(* Logix 5000 project; controller reports 1756-L63 rev 20.15; software revision 20.04; part 15 of 52 *)

        [677].log_data[17].valid := 1, [677].log_data[18].valid := 1, [677].log_data[19].valid := 1, [677].time.Year := 2023, [677].time.Month := 1, [677].time.Day := 12, [677].time.Minute := 49, [677].time.Second := 59, [678].log_data[0].min := 1.0, [678].log_data[0].max := 1.0, [678].log_data[0].total := 300.0, [678].log_data[0].time := 300.0, [678].log_data[0].minminute := 50, [678].log_data[0].maxminute := 50, [678].log_data[0].valid := 1, [678].log_data[1].valid := 1, [678].log_data[2].valid := 1, [678].log_data[3].valid := 1, [678].log_data[4].valid := 1, [678].log_data[5].valid := 1, [678].log_data[6].valid := 1, [678].log_data[7].valid := 1, [678].log_data[8].valid := 1, [678].log_data[9].valid := 1, [678].log_data[10].valid := 1, [678].log_data[11].valid := 1, [678].log_data[12].valid := 1, [678].log_data[13].valid := 1, [678].log_data[14].valid := 1, [678].log_data[15].valid := 1, [678].log_data[16].valid := 1, [678].log_data[17].valid := 1, [678].log_data[18].valid := 1, [678].log_data[19].valid := 1, [678].time.Year := 2023, [678].time.Month := 1, [678].time.Day := 12, [678].time.Minute := 54, [678].time.Second := 59, [679].log_data[0].min := 1.0, [679].log_data[0].max := 1.0, [679].log_data[0].total := 300.0, [679].log_data[0].time := 300.0, [679].log_data[0].minminute := 55, [679].log_data[0].maxminute := 55, [679].log_data[0].valid := 1, [679].log_data[1].valid := 1, [679].log_data[2].valid := 1, [679].log_data[3].valid := 1, [679].log_data[4].valid := 1, [679].log_data[5].valid := 1, [679].log_data[6].valid := 1, [679].log_data[7].valid := 1, [679].log_data[8].valid := 1, [679].log_data[9].valid := 1, [679].log_data[10].valid := 1, [679].log_data[11].valid := 1, [679].log_data[12].valid := 1, [679].log_data[13].valid := 1, [679].log_data[14].valid := 1,
        [679].log_data[15].valid := 1, [679].log_data[16].valid := 1, [679].log_data[17].valid := 1, [679].log_data[18].valid := 1, [679].log_data[19].valid := 1, [679].time.Year := 2023, [679].time.Month := 1, [679].time.Day := 12, [679].time.Minute := 59, [679].time.Second := 59, [680].log_data[0].min := 1.0, [680].log_data[0].max := 1.0, [680].log_data[0].total := 299.5, [680].log_data[0].time := 299.5, [680].log_data[0].valid := 1, [680].log_data[1].valid := 1, [680].log_data[2].valid := 1, [680].log_data[3].valid := 1, [680].log_data[4].valid := 1, [680].log_data[5].valid := 1, [680].log_data[6].valid := 1, [680].log_data[7].valid := 1, [680].log_data[8].valid := 1, [680].log_data[9].valid := 1, [680].log_data[10].valid := 1, [680].log_data[11].valid := 1, [680].log_data[12].valid := 1, [680].log_data[13].valid := 1, [680].log_data[14].valid := 1, [680].log_data[15].valid := 1, [680].log_data[16].valid := 1, [680].log_data[17].valid := 1, [680].log_data[18].valid := 1, [680].log_data[19].valid := 1, [680].time.Year := 2023, [680].time.Month := 1, [680].time.Day := 12, [680].time.Hour := 1, [680].time.Minute := 4, [680].time.Second := 59, [681].log_data[0].min := 1.0, [681].log_data[0].max := 1.0, [681].log_data[0].total := 300.0, [681].log_data[0].time := 300.0, [681].log_data[0].minminute := 5, [681].log_data[0].maxminute := 5, [681].log_data[0].valid := 1, [681].log_data[1].valid := 1, [681].log_data[2].valid := 1, [681].log_data[3].valid := 1, [681].log_data[4].valid := 1, [681].log_data[5].valid := 1, [681].log_data[6].valid := 1, [681].log_data[7].valid := 1, [681].log_data[8].valid := 1, [681].log_data[9].valid := 1, [681].log_data[10].valid := 1, [681].log_data[11].valid := 1, [681].log_data[12].valid := 1, [681].log_data[13].valid := 1,
        [681].log_data[14].valid := 1, [681].log_data[15].valid := 1, [681].log_data[16].valid := 1, [681].log_data[17].valid := 1, [681].log_data[18].valid := 1, [681].log_data[19].valid := 1, [681].time.Year := 2023, [681].time.Month := 1, [681].time.Day := 12, [681].time.Hour := 1, [681].time.Minute := 9, [681].time.Second := 59, [682].log_data[0].min := 1.0, [682].log_data[0].max := 1.0, [682].log_data[0].total := 300.0, [682].log_data[0].time := 300.0, [682].log_data[0].minminute := 10, [682].log_data[0].maxminute := 10, [682].log_data[0].valid := 1, [682].log_data[1].valid := 1, [682].log_data[2].valid := 1, [682].log_data[3].valid := 1, [682].log_data[4].valid := 1, [682].log_data[5].valid := 1, [682].log_data[6].valid := 1, [682].log_data[7].valid := 1, [682].log_data[8].valid := 1, [682].log_data[9].valid := 1, [682].log_data[10].valid := 1, [682].log_data[11].valid := 1, [682].log_data[12].valid := 1, [682].log_data[13].valid := 1, [682].log_data[14].valid := 1, [682].log_data[15].valid := 1, [682].log_data[16].valid := 1, [682].log_data[17].valid := 1, [682].log_data[18].valid := 1, [682].log_data[19].valid := 1, [682].time.Year := 2023, [682].time.Month := 1, [682].time.Day := 12, [682].time.Hour := 1, [682].time.Minute := 14, [682].time.Second := 59, [683].log_data[0].min := 1.0, [683].log_data[0].max := 1.0, [683].log_data[0].total := 300.0, [683].log_data[0].time := 300.0, [683].log_data[0].minminute := 15, [683].log_data[0].maxminute := 15, [683].log_data[0].valid := 1, [683].log_data[1].valid := 1, [683].log_data[2].valid := 1, [683].log_data[3].valid := 1, [683].log_data[4].valid := 1, [683].log_data[5].valid := 1, [683].log_data[6].valid := 1, [683].log_data[7].valid := 1, [683].log_data[8].valid := 1, [683].log_data[9].valid := 1,
        [683].log_data[10].valid := 1, [683].log_data[11].valid := 1, [683].log_data[12].valid := 1, [683].log_data[13].valid := 1, [683].log_data[14].valid := 1, [683].log_data[15].valid := 1, [683].log_data[16].valid := 1, [683].log_data[17].valid := 1, [683].log_data[18].valid := 1, [683].log_data[19].valid := 1, [683].time.Year := 2023, [683].time.Month := 1, [683].time.Day := 12, [683].time.Hour := 1, [683].time.Minute := 19, [683].time.Second := 59, [684].log_data[0].min := 1.0, [684].log_data[0].max := 1.0, [684].log_data[0].total := 300.0, [684].log_data[0].time := 300.0, [684].log_data[0].minminute := 20, [684].log_data[0].maxminute := 20, [684].log_data[0].valid := 1, [684].log_data[1].valid := 1, [684].log_data[2].valid := 1, [684].log_data[3].valid := 1, [684].log_data[4].valid := 1, [684].log_data[5].valid := 1, [684].log_data[6].valid := 1, [684].log_data[7].valid := 1, [684].log_data[8].valid := 1, [684].log_data[9].valid := 1, [684].log_data[10].valid := 1, [684].log_data[11].valid := 1, [684].log_data[12].valid := 1, [684].log_data[13].valid := 1, [684].log_data[14].valid := 1, [684].log_data[15].valid := 1, [684].log_data[16].valid := 1, [684].log_data[17].valid := 1, [684].log_data[18].valid := 1, [684].log_data[19].valid := 1, [684].time.Year := 2023, [684].time.Month := 1, [684].time.Day := 12, [684].time.Hour := 1, [684].time.Minute := 24, [684].time.Second := 59, [685].log_data[0].min := 1.0, [685].log_data[0].max := 1.0, [685].log_data[0].total := 300.0, [685].log_data[0].time := 300.0, [685].log_data[0].minminute := 25, [685].log_data[0].maxminute := 25, [685].log_data[0].valid := 1, [685].log_data[1].valid := 1, [685].log_data[2].valid := 1, [685].log_data[3].valid := 1, [685].log_data[4].valid := 1, [685].log_data[5].valid := 1,
        [685].log_data[6].valid := 1, [685].log_data[7].valid := 1, [685].log_data[8].valid := 1, [685].log_data[9].valid := 1, [685].log_data[10].valid := 1, [685].log_data[11].valid := 1, [685].log_data[12].valid := 1, [685].log_data[13].valid := 1, [685].log_data[14].valid := 1, [685].log_data[15].valid := 1, [685].log_data[16].valid := 1, [685].log_data[17].valid := 1, [685].log_data[18].valid := 1, [685].log_data[19].valid := 1, [685].time.Year := 2023, [685].time.Month := 1, [685].time.Day := 12, [685].time.Hour := 1, [685].time.Minute := 29, [685].time.Second := 59, [686].log_data[0].min := 1.0, [686].log_data[0].max := 1.0, [686].log_data[0].total := 300.0, [686].log_data[0].time := 300.0, [686].log_data[0].minminute := 30, [686].log_data[0].maxminute := 30, [686].log_data[0].valid := 1, [686].log_data[1].valid := 1, [686].log_data[2].valid := 1, [686].log_data[3].valid := 1, [686].log_data[4].valid := 1, [686].log_data[5].valid := 1, [686].log_data[6].valid := 1, [686].log_data[7].valid := 1, [686].log_data[8].valid := 1, [686].log_data[9].valid := 1, [686].log_data[10].valid := 1, [686].log_data[11].valid := 1, [686].log_data[12].valid := 1, [686].log_data[13].valid := 1, [686].log_data[14].valid := 1, [686].log_data[15].valid := 1, [686].log_data[16].valid := 1, [686].log_data[17].valid := 1, [686].log_data[18].valid := 1, [686].log_data[19].valid := 1, [686].time.Year := 2023, [686].time.Month := 1, [686].time.Day := 12, [686].time.Hour := 1, [686].time.Minute := 34, [686].time.Second := 59, [687].log_data[0].min := 1.0, [687].log_data[0].max := 1.0, [687].log_data[0].total := 300.0, [687].log_data[0].time := 300.0, [687].log_data[0].minminute := 35, [687].log_data[0].maxminute := 35, [687].log_data[0].valid := 1, [687].log_data[1].valid := 1,
        [687].log_data[2].valid := 1, [687].log_data[3].valid := 1, [687].log_data[4].valid := 1, [687].log_data[5].valid := 1, [687].log_data[6].valid := 1, [687].log_data[7].valid := 1, [687].log_data[8].valid := 1, [687].log_data[9].valid := 1, [687].log_data[10].valid := 1, [687].log_data[11].valid := 1, [687].log_data[12].valid := 1, [687].log_data[13].valid := 1, [687].log_data[14].valid := 1, [687].log_data[15].valid := 1, [687].log_data[16].valid := 1, [687].log_data[17].valid := 1, [687].log_data[18].valid := 1, [687].log_data[19].valid := 1, [687].time.Year := 2023, [687].time.Month := 1, [687].time.Day := 12, [687].time.Hour := 1, [687].time.Minute := 39, [687].time.Second := 59, [688].log_data[0].min := 1.0, [688].log_data[0].max := 1.0, [688].log_data[0].total := 300.0, [688].log_data[0].time := 300.0, [688].log_data[0].minminute := 40, [688].log_data[0].maxminute := 40, [688].log_data[0].valid := 1, [688].log_data[1].valid := 1, [688].log_data[2].valid := 1, [688].log_data[3].valid := 1, [688].log_data[4].valid := 1, [688].log_data[5].valid := 1, [688].log_data[6].valid := 1, [688].log_data[7].valid := 1, [688].log_data[8].valid := 1, [688].log_data[9].valid := 1, [688].log_data[10].valid := 1, [688].log_data[11].valid := 1, [688].log_data[12].valid := 1, [688].log_data[13].valid := 1, [688].log_data[14].valid := 1, [688].log_data[15].valid := 1, [688].log_data[16].valid := 1, [688].log_data[17].valid := 1, [688].log_data[18].valid := 1, [688].log_data[19].valid := 1, [688].time.Year := 2023, [688].time.Month := 1, [688].time.Day := 12, [688].time.Hour := 1, [688].time.Minute := 44, [688].time.Second := 59, [689].log_data[0].min := 1.0, [689].log_data[0].max := 1.0, [689].log_data[0].total := 300.0, [689].log_data[0].time := 300.0,
        [689].log_data[0].minminute := 45, [689].log_data[0].maxminute := 45, [689].log_data[0].valid := 1, [689].log_data[1].valid := 1, [689].log_data[2].valid := 1, [689].log_data[3].valid := 1, [689].log_data[4].valid := 1, [689].log_data[5].valid := 1, [689].log_data[6].valid := 1, [689].log_data[7].valid := 1, [689].log_data[8].valid := 1, [689].log_data[9].valid := 1, [689].log_data[10].valid := 1, [689].log_data[11].valid := 1, [689].log_data[12].valid := 1, [689].log_data[13].valid := 1, [689].log_data[14].valid := 1, [689].log_data[15].valid := 1, [689].log_data[16].valid := 1, [689].log_data[17].valid := 1, [689].log_data[18].valid := 1, [689].log_data[19].valid := 1, [689].time.Year := 2023, [689].time.Month := 1, [689].time.Day := 12, [689].time.Hour := 1, [689].time.Minute := 49, [689].time.Second := 59, [690].log_data[0].min := 1.0, [690].log_data[0].max := 1.0, [690].log_data[0].total := 300.0, [690].log_data[0].time := 300.0, [690].log_data[0].minminute := 50, [690].log_data[0].maxminute := 50, [690].log_data[0].valid := 1, [690].log_data[1].valid := 1, [690].log_data[2].valid := 1, [690].log_data[3].valid := 1, [690].log_data[4].valid := 1, [690].log_data[5].valid := 1, [690].log_data[6].valid := 1, [690].log_data[7].valid := 1, [690].log_data[8].valid := 1, [690].log_data[9].valid := 1, [690].log_data[10].valid := 1, [690].log_data[11].valid := 1, [690].log_data[12].valid := 1, [690].log_data[13].valid := 1, [690].log_data[14].valid := 1, [690].log_data[15].valid := 1, [690].log_data[16].valid := 1, [690].log_data[17].valid := 1, [690].log_data[18].valid := 1, [690].log_data[19].valid := 1, [690].time.Year := 2023, [690].time.Month := 1, [690].time.Day := 12, [690].time.Hour := 1, [690].time.Minute := 54, [690].time.Second := 59,
        [691].log_data[0].min := 1.0, [691].log_data[0].max := 1.0, [691].log_data[0].total := 300.0, [691].log_data[0].time := 300.0, [691].log_data[0].minminute := 55, [691].log_data[0].maxminute := 55, [691].log_data[0].valid := 1, [691].log_data[1].valid := 1, [691].log_data[2].valid := 1, [691].log_data[3].valid := 1, [691].log_data[4].valid := 1, [691].log_data[5].valid := 1, [691].log_data[6].valid := 1, [691].log_data[7].valid := 1, [691].log_data[8].valid := 1, [691].log_data[9].valid := 1, [691].log_data[10].valid := 1, [691].log_data[11].valid := 1, [691].log_data[12].valid := 1, [691].log_data[13].valid := 1, [691].log_data[14].valid := 1, [691].log_data[15].valid := 1, [691].log_data[16].valid := 1, [691].log_data[17].valid := 1, [691].log_data[18].valid := 1, [691].log_data[19].valid := 1, [691].time.Year := 2023, [691].time.Month := 1, [691].time.Day := 12, [691].time.Hour := 1, [691].time.Minute := 59, [691].time.Second := 59, [692].log_data[0].min := 1.0, [692].log_data[0].max := 1.0, [692].log_data[0].total := 300.0, [692].log_data[0].time := 300.0, [692].log_data[0].valid := 1, [692].log_data[1].valid := 1, [692].log_data[2].valid := 1, [692].log_data[3].valid := 1, [692].log_data[4].valid := 1, [692].log_data[5].valid := 1, [692].log_data[6].valid := 1, [692].log_data[7].valid := 1, [692].log_data[8].valid := 1, [692].log_data[9].valid := 1, [692].log_data[10].valid := 1, [692].log_data[11].valid := 1, [692].log_data[12].valid := 1, [692].log_data[13].valid := 1, [692].log_data[14].valid := 1, [692].log_data[15].valid := 1, [692].log_data[16].valid := 1, [692].log_data[17].valid := 1, [692].log_data[18].valid := 1, [692].log_data[19].valid := 1, [692].time.Year := 2023, [692].time.Month := 1, [692].time.Day := 12, [692].time.Hour := 2,
        [692].time.Minute := 4, [692].time.Second := 59, [693].log_data[0].min := 1.0, [693].log_data[0].max := 1.0, [693].log_data[0].total := 300.0, [693].log_data[0].time := 300.0, [693].log_data[0].minminute := 5, [693].log_data[0].maxminute := 5, [693].log_data[0].valid := 1, [693].log_data[1].valid := 1, [693].log_data[2].valid := 1, [693].log_data[3].valid := 1, [693].log_data[4].valid := 1, [693].log_data[5].valid := 1, [693].log_data[6].valid := 1, [693].log_data[7].valid := 1, [693].log_data[8].valid := 1, [693].log_data[9].valid := 1, [693].log_data[10].valid := 1, [693].log_data[11].valid := 1, [693].log_data[12].valid := 1, [693].log_data[13].valid := 1, [693].log_data[14].valid := 1, [693].log_data[15].valid := 1, [693].log_data[16].valid := 1, [693].log_data[17].valid := 1, [693].log_data[18].valid := 1, [693].log_data[19].valid := 1, [693].time.Year := 2023, [693].time.Month := 1, [693].time.Day := 12, [693].time.Hour := 2, [693].time.Minute := 9, [693].time.Second := 59, [694].log_data[0].min := 1.0, [694].log_data[0].max := 1.0, [694].log_data[0].total := 300.0, [694].log_data[0].time := 300.0, [694].log_data[0].minminute := 10, [694].log_data[0].maxminute := 10, [694].log_data[0].valid := 1, [694].log_data[1].valid := 1, [694].log_data[2].valid := 1, [694].log_data[3].valid := 1, [694].log_data[4].valid := 1, [694].log_data[5].valid := 1, [694].log_data[6].valid := 1, [694].log_data[7].valid := 1, [694].log_data[8].valid := 1, [694].log_data[9].valid := 1, [694].log_data[10].valid := 1, [694].log_data[11].valid := 1, [694].log_data[12].valid := 1, [694].log_data[13].valid := 1, [694].log_data[14].valid := 1, [694].log_data[15].valid := 1, [694].log_data[16].valid := 1, [694].log_data[17].valid := 1, [694].log_data[18].valid := 1, [694].log_data[19].valid := 1,
        [694].time.Year := 2023, [694].time.Month := 1, [694].time.Day := 12, [694].time.Hour := 2, [694].time.Minute := 14, [694].time.Second := 59, [695].log_data[0].min := 1.0, [695].log_data[0].max := 1.0, [695].log_data[0].total := 300.0, [695].log_data[0].time := 300.0, [695].log_data[0].minminute := 15, [695].log_data[0].maxminute := 15, [695].log_data[0].valid := 1, [695].log_data[1].valid := 1, [695].log_data[2].valid := 1, [695].log_data[3].valid := 1, [695].log_data[4].valid := 1, [695].log_data[5].valid := 1, [695].log_data[6].valid := 1, [695].log_data[7].valid := 1, [695].log_data[8].valid := 1, [695].log_data[9].valid := 1, [695].log_data[10].valid := 1, [695].log_data[11].valid := 1, [695].log_data[12].valid := 1, [695].log_data[13].valid := 1, [695].log_data[14].valid := 1, [695].log_data[15].valid := 1, [695].log_data[16].valid := 1, [695].log_data[17].valid := 1, [695].log_data[18].valid := 1, [695].log_data[19].valid := 1, [695].time.Year := 2023, [695].time.Month := 1, [695].time.Day := 12, [695].time.Hour := 2, [695].time.Minute := 19, [695].time.Second := 59, [696].log_data[0].min := 1.0, [696].log_data[0].max := 1.0, [696].log_data[0].total := 300.0, [696].log_data[0].time := 300.0, [696].log_data[0].minminute := 20, [696].log_data[0].maxminute := 20, [696].log_data[0].valid := 1, [696].log_data[1].valid := 1, [696].log_data[2].valid := 1, [696].log_data[3].valid := 1, [696].log_data[4].valid := 1, [696].log_data[5].valid := 1, [696].log_data[6].valid := 1, [696].log_data[7].valid := 1, [696].log_data[8].valid := 1, [696].log_data[9].valid := 1, [696].log_data[10].valid := 1, [696].log_data[11].valid := 1, [696].log_data[12].valid := 1, [696].log_data[13].valid := 1, [696].log_data[14].valid := 1, [696].log_data[15].valid := 1,
        [696].log_data[16].valid := 1, [696].log_data[17].valid := 1, [696].log_data[18].valid := 1, [696].log_data[19].valid := 1, [696].time.Year := 2023, [696].time.Month := 1, [696].time.Day := 12, [696].time.Hour := 2, [696].time.Minute := 24, [696].time.Second := 59, [697].log_data[0].min := 1.0, [697].log_data[0].max := 1.0, [697].log_data[0].total := 300.0, [697].log_data[0].time := 300.0, [697].log_data[0].minminute := 25, [697].log_data[0].maxminute := 25, [697].log_data[0].valid := 1, [697].log_data[1].valid := 1, [697].log_data[2].valid := 1, [697].log_data[3].valid := 1, [697].log_data[4].valid := 1, [697].log_data[5].valid := 1, [697].log_data[6].valid := 1, [697].log_data[7].valid := 1, [697].log_data[8].valid := 1, [697].log_data[9].valid := 1, [697].log_data[10].valid := 1, [697].log_data[11].valid := 1, [697].log_data[12].valid := 1, [697].log_data[13].valid := 1, [697].log_data[14].valid := 1, [697].log_data[15].valid := 1, [697].log_data[16].valid := 1, [697].log_data[17].valid := 1, [697].log_data[18].valid := 1, [697].log_data[19].valid := 1, [697].time.Year := 2023, [697].time.Month := 1, [697].time.Day := 12, [697].time.Hour := 2, [697].time.Minute := 29, [697].time.Second := 59, [698].log_data[0].min := 1.0, [698].log_data[0].max := 1.0, [698].log_data[0].total := 300.0, [698].log_data[0].time := 300.0, [698].log_data[0].minminute := 30, [698].log_data[0].maxminute := 30, [698].log_data[0].valid := 1, [698].log_data[1].valid := 1, [698].log_data[2].valid := 1, [698].log_data[3].valid := 1, [698].log_data[4].valid := 1, [698].log_data[5].valid := 1, [698].log_data[6].valid := 1, [698].log_data[7].valid := 1, [698].log_data[8].valid := 1, [698].log_data[9].valid := 1, [698].log_data[10].valid := 1, [698].log_data[11].valid := 1,
        [698].log_data[12].valid := 1, [698].log_data[13].valid := 1, [698].log_data[14].valid := 1, [698].log_data[15].valid := 1, [698].log_data[16].valid := 1, [698].log_data[17].valid := 1, [698].log_data[18].valid := 1, [698].log_data[19].valid := 1, [698].time.Year := 2023, [698].time.Month := 1, [698].time.Day := 12, [698].time.Hour := 2, [698].time.Minute := 34, [698].time.Second := 59, [699].log_data[0].min := 1.0, [699].log_data[0].max := 1.0, [699].log_data[0].total := 300.0, [699].log_data[0].time := 300.0, [699].log_data[0].minminute := 35, [699].log_data[0].maxminute := 35, [699].log_data[0].valid := 1, [699].log_data[1].valid := 1, [699].log_data[2].valid := 1, [699].log_data[3].valid := 1, [699].log_data[4].valid := 1, [699].log_data[5].valid := 1, [699].log_data[6].valid := 1, [699].log_data[7].valid := 1, [699].log_data[8].valid := 1, [699].log_data[9].valid := 1, [699].log_data[10].valid := 1, [699].log_data[11].valid := 1, [699].log_data[12].valid := 1, [699].log_data[13].valid := 1, [699].log_data[14].valid := 1, [699].log_data[15].valid := 1, [699].log_data[16].valid := 1, [699].log_data[17].valid := 1, [699].log_data[18].valid := 1, [699].log_data[19].valid := 1, [699].time.Year := 2023, [699].time.Month := 1, [699].time.Day := 12, [699].time.Hour := 2, [699].time.Minute := 39, [699].time.Second := 59, [700].log_data[0].min := 1.0, [700].log_data[0].max := 1.0, [700].log_data[0].total := 300.0, [700].log_data[0].time := 300.0, [700].log_data[0].minminute := 40, [700].log_data[0].maxminute := 40, [700].log_data[0].valid := 1, [700].log_data[1].valid := 1, [700].log_data[2].valid := 1, [700].log_data[3].valid := 1, [700].log_data[4].valid := 1, [700].log_data[5].valid := 1, [700].log_data[6].valid := 1, [700].log_data[7].valid := 1,
        [700].log_data[8].valid := 1, [700].log_data[9].valid := 1, [700].log_data[10].valid := 1, [700].log_data[11].valid := 1, [700].log_data[12].valid := 1, [700].log_data[13].valid := 1, [700].log_data[14].valid := 1, [700].log_data[15].valid := 1, [700].log_data[16].valid := 1, [700].log_data[17].valid := 1, [700].log_data[18].valid := 1, [700].log_data[19].valid := 1, [700].time.Year := 2023, [700].time.Month := 1, [700].time.Day := 12, [700].time.Hour := 2, [700].time.Minute := 44, [700].time.Second := 59, [701].log_data[0].min := 1.0, [701].log_data[0].max := 1.0, [701].log_data[0].total := 300.0, [701].log_data[0].time := 300.0, [701].log_data[0].minminute := 45, [701].log_data[0].maxminute := 45, [701].log_data[0].valid := 1, [701].log_data[1].valid := 1, [701].log_data[2].valid := 1, [701].log_data[3].valid := 1, [701].log_data[4].valid := 1, [701].log_data[5].valid := 1, [701].log_data[6].valid := 1, [701].log_data[7].valid := 1, [701].log_data[8].valid := 1, [701].log_data[9].valid := 1, [701].log_data[10].valid := 1, [701].log_data[11].valid := 1, [701].log_data[12].valid := 1, [701].log_data[13].valid := 1, [701].log_data[14].valid := 1, [701].log_data[15].valid := 1, [701].log_data[16].valid := 1, [701].log_data[17].valid := 1, [701].log_data[18].valid := 1, [701].log_data[19].valid := 1, [701].time.Year := 2023, [701].time.Month := 1, [701].time.Day := 12, [701].time.Hour := 2, [701].time.Minute := 49, [701].time.Second := 59, [702].log_data[0].min := 1.0, [702].log_data[0].max := 1.0, [702].log_data[0].total := 300.0, [702].log_data[0].time := 300.0, [702].log_data[0].minminute := 50, [702].log_data[0].maxminute := 50, [702].log_data[0].valid := 1, [702].log_data[1].valid := 1, [702].log_data[2].valid := 1, [702].log_data[3].valid := 1,
        [702].log_data[4].valid := 1, [702].log_data[5].valid := 1, [702].log_data[6].valid := 1, [702].log_data[7].valid := 1, [702].log_data[8].valid := 1, [702].log_data[9].valid := 1, [702].log_data[10].valid := 1, [702].log_data[11].valid := 1, [702].log_data[12].valid := 1, [702].log_data[13].valid := 1, [702].log_data[14].valid := 1, [702].log_data[15].valid := 1, [702].log_data[16].valid := 1, [702].log_data[17].valid := 1, [702].log_data[18].valid := 1, [702].log_data[19].valid := 1, [702].time.Year := 2023, [702].time.Month := 1, [702].time.Day := 12, [702].time.Hour := 2, [702].time.Minute := 54, [702].time.Second := 59, [703].log_data[0].min := 1.0, [703].log_data[0].max := 1.0, [703].log_data[0].total := 300.0, [703].log_data[0].time := 300.0, [703].log_data[0].minminute := 55, [703].log_data[0].maxminute := 55, [703].log_data[0].valid := 1, [703].log_data[1].valid := 1, [703].log_data[2].valid := 1, [703].log_data[3].valid := 1, [703].log_data[4].valid := 1, [703].log_data[5].valid := 1, [703].log_data[6].valid := 1, [703].log_data[7].valid := 1, [703].log_data[8].valid := 1, [703].log_data[9].valid := 1, [703].log_data[10].valid := 1, [703].log_data[11].valid := 1, [703].log_data[12].valid := 1, [703].log_data[13].valid := 1, [703].log_data[14].valid := 1, [703].log_data[15].valid := 1, [703].log_data[16].valid := 1, [703].log_data[17].valid := 1, [703].log_data[18].valid := 1, [703].log_data[19].valid := 1, [703].time.Year := 2023, [703].time.Month := 1, [703].time.Day := 12, [703].time.Hour := 2, [703].time.Minute := 59, [703].time.Second := 59, [704].log_data[0].min := 1.0, [704].log_data[0].max := 1.0, [704].log_data[0].total := 300.0, [704].log_data[0].time := 300.0, [704].log_data[0].valid := 1, [704].log_data[1].valid := 1,
        [704].log_data[2].valid := 1, [704].log_data[3].valid := 1, [704].log_data[4].valid := 1, [704].log_data[5].valid := 1, [704].log_data[6].valid := 1, [704].log_data[7].valid := 1, [704].log_data[8].valid := 1, [704].log_data[9].valid := 1, [704].log_data[10].valid := 1, [704].log_data[11].valid := 1, [704].log_data[12].valid := 1, [704].log_data[13].valid := 1, [704].log_data[14].valid := 1, [704].log_data[15].valid := 1, [704].log_data[16].valid := 1, [704].log_data[17].valid := 1, [704].log_data[18].valid := 1, [704].log_data[19].valid := 1, [704].time.Year := 2023, [704].time.Month := 1, [704].time.Day := 12, [704].time.Hour := 3, [704].time.Minute := 4, [704].time.Second := 59, [705].log_data[0].min := 1.0, [705].log_data[0].max := 1.0, [705].log_data[0].total := 300.0, [705].log_data[0].time := 300.0, [705].log_data[0].minminute := 5, [705].log_data[0].maxminute := 5, [705].log_data[0].valid := 1, [705].log_data[1].valid := 1, [705].log_data[2].valid := 1, [705].log_data[3].valid := 1, [705].log_data[4].valid := 1, [705].log_data[5].valid := 1, [705].log_data[6].valid := 1, [705].log_data[7].valid := 1, [705].log_data[8].valid := 1, [705].log_data[9].valid := 1, [705].log_data[10].valid := 1, [705].log_data[11].valid := 1, [705].log_data[12].valid := 1, [705].log_data[13].valid := 1, [705].log_data[14].valid := 1, [705].log_data[15].valid := 1, [705].log_data[16].valid := 1, [705].log_data[17].valid := 1, [705].log_data[18].valid := 1, [705].log_data[19].valid := 1, [705].time.Year := 2023, [705].time.Month := 1, [705].time.Day := 12, [705].time.Hour := 3, [705].time.Minute := 9, [705].time.Second := 59, [706].log_data[0].min := 1.0, [706].log_data[0].max := 1.0, [706].log_data[0].total := 300.0, [706].log_data[0].time := 300.0,
        [706].log_data[0].minminute := 10, [706].log_data[0].maxminute := 10, [706].log_data[0].valid := 1, [706].log_data[1].valid := 1, [706].log_data[2].valid := 1, [706].log_data[3].valid := 1, [706].log_data[4].valid := 1, [706].log_data[5].valid := 1, [706].log_data[6].valid := 1, [706].log_data[7].valid := 1, [706].log_data[8].valid := 1, [706].log_data[9].valid := 1, [706].log_data[10].valid := 1, [706].log_data[11].valid := 1, [706].log_data[12].valid := 1, [706].log_data[13].valid := 1, [706].log_data[14].valid := 1, [706].log_data[15].valid := 1, [706].log_data[16].valid := 1, [706].log_data[17].valid := 1, [706].log_data[18].valid := 1, [706].log_data[19].valid := 1, [706].time.Year := 2023, [706].time.Month := 1, [706].time.Day := 12, [706].time.Hour := 3, [706].time.Minute := 14, [706].time.Second := 59, [707].log_data[0].min := 1.0, [707].log_data[0].max := 1.0, [707].log_data[0].total := 300.0, [707].log_data[0].time := 300.0, [707].log_data[0].minminute := 15, [707].log_data[0].maxminute := 15, [707].log_data[0].valid := 1, [707].log_data[1].valid := 1, [707].log_data[2].valid := 1, [707].log_data[3].valid := 1, [707].log_data[4].valid := 1, [707].log_data[5].valid := 1, [707].log_data[6].valid := 1, [707].log_data[7].valid := 1, [707].log_data[8].valid := 1, [707].log_data[9].valid := 1, [707].log_data[10].valid := 1, [707].log_data[11].valid := 1, [707].log_data[12].valid := 1, [707].log_data[13].valid := 1, [707].log_data[14].valid := 1, [707].log_data[15].valid := 1, [707].log_data[16].valid := 1, [707].log_data[17].valid := 1, [707].log_data[18].valid := 1, [707].log_data[19].valid := 1, [707].time.Year := 2023, [707].time.Month := 1, [707].time.Day := 12, [707].time.Hour := 3, [707].time.Minute := 19, [707].time.Second := 59,
        [708].log_data[0].min := 1.0, [708].log_data[0].max := 1.0, [708].log_data[0].total := 300.0, [708].log_data[0].time := 300.0, [708].log_data[0].minminute := 20, [708].log_data[0].maxminute := 20, [708].log_data[0].valid := 1, [708].log_data[1].valid := 1, [708].log_data[2].valid := 1, [708].log_data[3].valid := 1, [708].log_data[4].valid := 1, [708].log_data[5].valid := 1, [708].log_data[6].valid := 1, [708].log_data[7].valid := 1, [708].log_data[8].valid := 1, [708].log_data[9].valid := 1, [708].log_data[10].valid := 1, [708].log_data[11].valid := 1, [708].log_data[12].valid := 1, [708].log_data[13].valid := 1, [708].log_data[14].valid := 1, [708].log_data[15].valid := 1, [708].log_data[16].valid := 1, [708].log_data[17].valid := 1, [708].log_data[18].valid := 1, [708].log_data[19].valid := 1, [708].time.Year := 2023, [708].time.Month := 1, [708].time.Day := 12, [708].time.Hour := 3, [708].time.Minute := 24, [708].time.Second := 59, [709].log_data[0].min := 1.0, [709].log_data[0].max := 1.0, [709].log_data[0].total := 300.0, [709].log_data[0].time := 300.0, [709].log_data[0].minminute := 25, [709].log_data[0].maxminute := 25, [709].log_data[0].valid := 1, [709].log_data[1].valid := 1, [709].log_data[2].valid := 1, [709].log_data[3].valid := 1, [709].log_data[4].valid := 1, [709].log_data[5].valid := 1, [709].log_data[6].valid := 1, [709].log_data[7].valid := 1, [709].log_data[8].valid := 1, [709].log_data[9].valid := 1, [709].log_data[10].valid := 1, [709].log_data[11].valid := 1, [709].log_data[12].valid := 1, [709].log_data[13].valid := 1, [709].log_data[14].valid := 1, [709].log_data[15].valid := 1, [709].log_data[16].valid := 1, [709].log_data[17].valid := 1, [709].log_data[18].valid := 1, [709].log_data[19].valid := 1, [709].time.Year := 2023, [709].time.Month := 1,
        [709].time.Day := 12, [709].time.Hour := 3, [709].time.Minute := 29, [709].time.Second := 59, [710].log_data[0].min := 1.0, [710].log_data[0].max := 1.0, [710].log_data[0].total := 300.0, [710].log_data[0].time := 300.0, [710].log_data[0].minminute := 30, [710].log_data[0].maxminute := 30, [710].log_data[0].valid := 1, [710].log_data[1].valid := 1, [710].log_data[2].valid := 1, [710].log_data[3].valid := 1, [710].log_data[4].valid := 1, [710].log_data[5].valid := 1, [710].log_data[6].valid := 1, [710].log_data[7].valid := 1, [710].log_data[8].valid := 1, [710].log_data[9].valid := 1, [710].log_data[10].valid := 1, [710].log_data[11].valid := 1, [710].log_data[12].valid := 1, [710].log_data[13].valid := 1, [710].log_data[14].valid := 1, [710].log_data[15].valid := 1, [710].log_data[16].valid := 1, [710].log_data[17].valid := 1, [710].log_data[18].valid := 1, [710].log_data[19].valid := 1, [710].time.Year := 2023, [710].time.Month := 1, [710].time.Day := 12, [710].time.Hour := 3, [710].time.Minute := 34, [710].time.Second := 59, [711].log_data[0].min := 1.0, [711].log_data[0].max := 1.0, [711].log_data[0].total := 300.0, [711].log_data[0].time := 300.0, [711].log_data[0].minminute := 35, [711].log_data[0].maxminute := 35, [711].log_data[0].valid := 1, [711].log_data[1].valid := 1, [711].log_data[2].valid := 1, [711].log_data[3].valid := 1, [711].log_data[4].valid := 1, [711].log_data[5].valid := 1, [711].log_data[6].valid := 1, [711].log_data[7].valid := 1, [711].log_data[8].valid := 1, [711].log_data[9].valid := 1, [711].log_data[10].valid := 1, [711].log_data[11].valid := 1, [711].log_data[12].valid := 1, [711].log_data[13].valid := 1, [711].log_data[14].valid := 1, [711].log_data[15].valid := 1, [711].log_data[16].valid := 1, [711].log_data[17].valid := 1,
        [711].log_data[18].valid := 1, [711].log_data[19].valid := 1, [711].time.Year := 2023, [711].time.Month := 1, [711].time.Day := 12, [711].time.Hour := 3, [711].time.Minute := 39, [711].time.Second := 59, [712].log_data[0].min := 1.0, [712].log_data[0].max := 1.0, [712].log_data[0].total := 300.0, [712].log_data[0].time := 300.0, [712].log_data[0].minminute := 40, [712].log_data[0].maxminute := 40, [712].log_data[0].valid := 1, [712].log_data[1].valid := 1, [712].log_data[2].valid := 1, [712].log_data[3].valid := 1, [712].log_data[4].valid := 1, [712].log_data[5].valid := 1, [712].log_data[6].valid := 1, [712].log_data[7].valid := 1, [712].log_data[8].valid := 1, [712].log_data[9].valid := 1, [712].log_data[10].valid := 1, [712].log_data[11].valid := 1, [712].log_data[12].valid := 1, [712].log_data[13].valid := 1, [712].log_data[14].valid := 1, [712].log_data[15].valid := 1, [712].log_data[16].valid := 1, [712].log_data[17].valid := 1, [712].log_data[18].valid := 1, [712].log_data[19].valid := 1, [712].time.Year := 2023, [712].time.Month := 1, [712].time.Day := 12, [712].time.Hour := 3, [712].time.Minute := 44, [712].time.Second := 59, [713].log_data[0].min := 1.0, [713].log_data[0].max := 1.0, [713].log_data[0].total := 300.0, [713].log_data[0].time := 300.0, [713].log_data[0].minminute := 45, [713].log_data[0].maxminute := 45, [713].log_data[0].valid := 1, [713].log_data[1].valid := 1, [713].log_data[2].valid := 1, [713].log_data[3].valid := 1, [713].log_data[4].valid := 1, [713].log_data[5].valid := 1, [713].log_data[6].valid := 1, [713].log_data[7].valid := 1, [713].log_data[8].valid := 1, [713].log_data[9].valid := 1, [713].log_data[10].valid := 1, [713].log_data[11].valid := 1, [713].log_data[12].valid := 1, [713].log_data[13].valid := 1,
        [713].log_data[14].valid := 1, [713].log_data[15].valid := 1, [713].log_data[16].valid := 1, [713].log_data[17].valid := 1, [713].log_data[18].valid := 1, [713].log_data[19].valid := 1, [713].time.Year := 2023, [713].time.Month := 1, [713].time.Day := 12, [713].time.Hour := 3, [713].time.Minute := 49, [713].time.Second := 59, [714].log_data[0].min := 1.0, [714].log_data[0].max := 1.0, [714].log_data[0].total := 300.0, [714].log_data[0].time := 300.0, [714].log_data[0].minminute := 50, [714].log_data[0].maxminute := 50, [714].log_data[0].valid := 1, [714].log_data[1].valid := 1, [714].log_data[2].valid := 1, [714].log_data[3].valid := 1, [714].log_data[4].valid := 1, [714].log_data[5].valid := 1, [714].log_data[6].valid := 1, [714].log_data[7].valid := 1, [714].log_data[8].valid := 1, [714].log_data[9].valid := 1, [714].log_data[10].valid := 1, [714].log_data[11].valid := 1, [714].log_data[12].valid := 1, [714].log_data[13].valid := 1, [714].log_data[14].valid := 1, [714].log_data[15].valid := 1, [714].log_data[16].valid := 1, [714].log_data[17].valid := 1, [714].log_data[18].valid := 1, [714].log_data[19].valid := 1, [714].time.Year := 2023, [714].time.Month := 1, [714].time.Day := 12, [714].time.Hour := 3, [714].time.Minute := 54, [714].time.Second := 59, [715].log_data[0].min := 1.0, [715].log_data[0].max := 1.0, [715].log_data[0].total := 300.0, [715].log_data[0].time := 300.0, [715].log_data[0].minminute := 55, [715].log_data[0].maxminute := 55, [715].log_data[0].valid := 1, [715].log_data[1].valid := 1, [715].log_data[2].valid := 1, [715].log_data[3].valid := 1, [715].log_data[4].valid := 1, [715].log_data[5].valid := 1, [715].log_data[6].valid := 1, [715].log_data[7].valid := 1, [715].log_data[8].valid := 1, [715].log_data[9].valid := 1,
        [715].log_data[10].valid := 1, [715].log_data[11].valid := 1, [715].log_data[12].valid := 1, [715].log_data[13].valid := 1, [715].log_data[14].valid := 1, [715].log_data[15].valid := 1, [715].log_data[16].valid := 1, [715].log_data[17].valid := 1, [715].log_data[18].valid := 1, [715].log_data[19].valid := 1, [715].time.Year := 2023, [715].time.Month := 1, [715].time.Day := 12, [715].time.Hour := 3, [715].time.Minute := 59, [715].time.Second := 59, [716].log_data[0].min := 1.0, [716].log_data[0].max := 1.0, [716].log_data[0].total := 300.0, [716].log_data[0].time := 300.0, [716].log_data[0].valid := 1, [716].log_data[1].valid := 1, [716].log_data[2].valid := 1, [716].log_data[3].valid := 1, [716].log_data[4].valid := 1, [716].log_data[5].valid := 1, [716].log_data[6].valid := 1, [716].log_data[7].valid := 1, [716].log_data[8].valid := 1, [716].log_data[9].valid := 1, [716].log_data[10].valid := 1, [716].log_data[11].valid := 1, [716].log_data[12].valid := 1, [716].log_data[13].valid := 1, [716].log_data[14].valid := 1, [716].log_data[15].valid := 1, [716].log_data[16].valid := 1, [716].log_data[17].valid := 1, [716].log_data[18].valid := 1, [716].log_data[19].valid := 1, [716].time.Year := 2023, [716].time.Month := 1, [716].time.Day := 12, [716].time.Hour := 4, [716].time.Minute := 4, [716].time.Second := 59, [717].log_data[0].min := 1.0, [717].log_data[0].max := 1.0, [717].log_data[0].total := 300.0, [717].log_data[0].time := 300.0, [717].log_data[0].minminute := 5, [717].log_data[0].maxminute := 5, [717].log_data[0].valid := 1, [717].log_data[1].valid := 1, [717].log_data[2].valid := 1, [717].log_data[3].valid := 1, [717].log_data[4].valid := 1, [717].log_data[5].valid := 1, [717].log_data[6].valid := 1, [717].log_data[7].valid := 1,
        [717].log_data[8].valid := 1, [717].log_data[9].valid := 1, [717].log_data[10].valid := 1, [717].log_data[11].valid := 1, [717].log_data[12].valid := 1, [717].log_data[13].valid := 1, [717].log_data[14].valid := 1, [717].log_data[15].valid := 1, [717].log_data[16].valid := 1, [717].log_data[17].valid := 1, [717].log_data[18].valid := 1, [717].log_data[19].valid := 1, [717].time.Year := 2023, [717].time.Month := 1, [717].time.Day := 12, [717].time.Hour := 4, [717].time.Minute := 9, [717].time.Second := 59, [718].log_data[0].min := 1.0, [718].log_data[0].max := 1.0, [718].log_data[0].total := 300.0, [718].log_data[0].time := 300.0, [718].log_data[0].minminute := 10, [718].log_data[0].maxminute := 10, [718].log_data[0].valid := 1, [718].log_data[1].valid := 1, [718].log_data[2].valid := 1, [718].log_data[3].valid := 1, [718].log_data[4].valid := 1, [718].log_data[5].valid := 1, [718].log_data[6].valid := 1, [718].log_data[7].valid := 1, [718].log_data[8].valid := 1, [718].log_data[9].valid := 1, [718].log_data[10].valid := 1, [718].log_data[11].valid := 1, [718].log_data[12].valid := 1, [718].log_data[13].valid := 1, [718].log_data[14].valid := 1, [718].log_data[15].valid := 1, [718].log_data[16].valid := 1, [718].log_data[17].valid := 1, [718].log_data[18].valid := 1, [718].log_data[19].valid := 1, [718].time.Year := 2023, [718].time.Month := 1, [718].time.Day := 12, [718].time.Hour := 4, [718].time.Minute := 14, [718].time.Second := 59, [719].log_data[0].min := 1.0, [719].log_data[0].max := 1.0, [719].log_data[0].total := 300.0, [719].log_data[0].time := 300.0, [719].log_data[0].minminute := 15, [719].log_data[0].maxminute := 15, [719].log_data[0].valid := 1, [719].log_data[1].valid := 1, [719].log_data[2].valid := 1, [719].log_data[3].valid := 1,
        [719].log_data[4].valid := 1, [719].log_data[5].valid := 1, [719].log_data[6].valid := 1, [719].log_data[7].valid := 1, [719].log_data[8].valid := 1, [719].log_data[9].valid := 1, [719].log_data[10].valid := 1, [719].log_data[11].valid := 1, [719].log_data[12].valid := 1, [719].log_data[13].valid := 1, [719].log_data[14].valid := 1, [719].log_data[15].valid := 1, [719].log_data[16].valid := 1, [719].log_data[17].valid := 1, [719].log_data[18].valid := 1, [719].log_data[19].valid := 1, [719].time.Year := 2023, [719].time.Month := 1, [719].time.Day := 12, [719].time.Hour := 4, [719].time.Minute := 19, [719].time.Second := 59, [720].log_data[0].min := 1.0, [720].log_data[0].max := 1.0, [720].log_data[0].total := 300.0, [720].log_data[0].time := 300.0, [720].log_data[0].minminute := 20, [720].log_data[0].maxminute := 20, [720].log_data[0].valid := 1, [720].log_data[1].valid := 1, [720].log_data[2].valid := 1, [720].log_data[3].valid := 1, [720].log_data[4].valid := 1, [720].log_data[5].valid := 1, [720].log_data[6].valid := 1, [720].log_data[7].valid := 1, [720].log_data[8].valid := 1, [720].log_data[9].valid := 1, [720].log_data[10].valid := 1, [720].log_data[11].valid := 1, [720].log_data[12].valid := 1, [720].log_data[13].valid := 1, [720].log_data[14].valid := 1, [720].log_data[15].valid := 1, [720].log_data[16].valid := 1, [720].log_data[17].valid := 1, [720].log_data[18].valid := 1, [720].log_data[19].valid := 1, [720].time.Year := 2023, [720].time.Month := 1, [720].time.Day := 12, [720].time.Hour := 4, [720].time.Minute := 24, [720].time.Second := 59, [721].log_data[0].min := 1.0, [721].log_data[0].max := 1.0, [721].log_data[0].total := 300.0, [721].log_data[0].time := 300.0, [721].log_data[0].minminute := 25, [721].log_data[0].maxminute := 25,
        [721].log_data[0].valid := 1, [721].log_data[1].valid := 1, [721].log_data[2].valid := 1, [721].log_data[3].valid := 1, [721].log_data[4].valid := 1, [721].log_data[5].valid := 1, [721].log_data[6].valid := 1, [721].log_data[7].valid := 1, [721].log_data[8].valid := 1, [721].log_data[9].valid := 1, [721].log_data[10].valid := 1, [721].log_data[11].valid := 1, [721].log_data[12].valid := 1, [721].log_data[13].valid := 1, [721].log_data[14].valid := 1, [721].log_data[15].valid := 1, [721].log_data[16].valid := 1, [721].log_data[17].valid := 1, [721].log_data[18].valid := 1, [721].log_data[19].valid := 1, [721].time.Year := 2023, [721].time.Month := 1, [721].time.Day := 12, [721].time.Hour := 4, [721].time.Minute := 29, [721].time.Second := 59, [722].log_data[0].min := 1.0, [722].log_data[0].max := 1.0, [722].log_data[0].total := 300.0, [722].log_data[0].time := 300.0, [722].log_data[0].minminute := 30, [722].log_data[0].maxminute := 30, [722].log_data[0].valid := 1, [722].log_data[1].valid := 1, [722].log_data[2].valid := 1, [722].log_data[3].valid := 1, [722].log_data[4].valid := 1, [722].log_data[5].valid := 1, [722].log_data[6].valid := 1, [722].log_data[7].valid := 1, [722].log_data[8].valid := 1, [722].log_data[9].valid := 1, [722].log_data[10].valid := 1, [722].log_data[11].valid := 1, [722].log_data[12].valid := 1, [722].log_data[13].valid := 1, [722].log_data[14].valid := 1, [722].log_data[15].valid := 1, [722].log_data[16].valid := 1, [722].log_data[17].valid := 1, [722].log_data[18].valid := 1, [722].log_data[19].valid := 1, [722].time.Year := 2023, [722].time.Month := 1, [722].time.Day := 12, [722].time.Hour := 4, [722].time.Minute := 34, [722].time.Second := 59, [723].log_data[0].min := 1.0, [723].log_data[0].max := 1.0,
        [723].log_data[0].total := 300.0, [723].log_data[0].time := 300.0, [723].log_data[0].minminute := 35, [723].log_data[0].maxminute := 35, [723].log_data[0].valid := 1, [723].log_data[1].valid := 1, [723].log_data[2].valid := 1, [723].log_data[3].valid := 1, [723].log_data[4].valid := 1, [723].log_data[5].valid := 1, [723].log_data[6].valid := 1, [723].log_data[7].valid := 1, [723].log_data[8].valid := 1, [723].log_data[9].valid := 1, [723].log_data[10].valid := 1, [723].log_data[11].valid := 1, [723].log_data[12].valid := 1, [723].log_data[13].valid := 1, [723].log_data[14].valid := 1, [723].log_data[15].valid := 1, [723].log_data[16].valid := 1, [723].log_data[17].valid := 1, [723].log_data[18].valid := 1, [723].log_data[19].valid := 1, [723].time.Year := 2023, [723].time.Month := 1, [723].time.Day := 12, [723].time.Hour := 4, [723].time.Minute := 39, [723].time.Second := 59, [724].log_data[0].min := 1.0, [724].log_data[0].max := 1.0, [724].log_data[0].total := 300.0, [724].log_data[0].time := 300.0, [724].log_data[0].minminute := 40, [724].log_data[0].maxminute := 40, [724].log_data[0].valid := 1, [724].log_data[1].valid := 1, [724].log_data[2].valid := 1, [724].log_data[3].valid := 1, [724].log_data[4].valid := 1, [724].log_data[5].valid := 1, [724].log_data[6].valid := 1, [724].log_data[7].valid := 1, [724].log_data[8].valid := 1, [724].log_data[9].valid := 1, [724].log_data[10].valid := 1, [724].log_data[11].valid := 1, [724].log_data[12].valid := 1, [724].log_data[13].valid := 1, [724].log_data[14].valid := 1, [724].log_data[15].valid := 1, [724].log_data[16].valid := 1, [724].log_data[17].valid := 1, [724].log_data[18].valid := 1, [724].log_data[19].valid := 1, [724].time.Year := 2023, [724].time.Month := 1, [724].time.Day := 12, [724].time.Hour := 4,
        [724].time.Minute := 44, [724].time.Second := 59, [725].log_data[0].min := 1.0, [725].log_data[0].max := 1.0, [725].log_data[0].total := 300.0, [725].log_data[0].time := 300.0, [725].log_data[0].minminute := 45, [725].log_data[0].maxminute := 45, [725].log_data[0].valid := 1, [725].log_data[1].valid := 1, [725].log_data[2].valid := 1, [725].log_data[3].valid := 1, [725].log_data[4].valid := 1, [725].log_data[5].valid := 1, [725].log_data[6].valid := 1, [725].log_data[7].valid := 1, [725].log_data[8].valid := 1, [725].log_data[9].valid := 1, [725].log_data[10].valid := 1, [725].log_data[11].valid := 1, [725].log_data[12].valid := 1, [725].log_data[13].valid := 1, [725].log_data[14].valid := 1, [725].log_data[15].valid := 1, [725].log_data[16].valid := 1, [725].log_data[17].valid := 1, [725].log_data[18].valid := 1, [725].log_data[19].valid := 1, [725].time.Year := 2023, [725].time.Month := 1, [725].time.Day := 12, [725].time.Hour := 4, [725].time.Minute := 49, [725].time.Second := 59, [726].log_data[0].min := 1.0, [726].log_data[0].max := 1.0, [726].log_data[0].total := 300.0, [726].log_data[0].time := 300.0, [726].log_data[0].minminute := 50, [726].log_data[0].maxminute := 50, [726].log_data[0].valid := 1, [726].log_data[1].valid := 1, [726].log_data[2].valid := 1, [726].log_data[3].valid := 1, [726].log_data[4].valid := 1, [726].log_data[5].valid := 1, [726].log_data[6].valid := 1, [726].log_data[7].valid := 1, [726].log_data[8].valid := 1, [726].log_data[9].valid := 1, [726].log_data[10].valid := 1, [726].log_data[11].valid := 1, [726].log_data[12].valid := 1, [726].log_data[13].valid := 1, [726].log_data[14].valid := 1, [726].log_data[15].valid := 1, [726].log_data[16].valid := 1, [726].log_data[17].valid := 1, [726].log_data[18].valid := 1, [726].log_data[19].valid := 1,
        [726].time.Year := 2023, [726].time.Month := 1, [726].time.Day := 12, [726].time.Hour := 4, [726].time.Minute := 54, [726].time.Second := 59, [727].log_data[0].min := 1.0, [727].log_data[0].max := 1.0, [727].log_data[0].total := 300.0, [727].log_data[0].time := 300.0, [727].log_data[0].minminute := 55, [727].log_data[0].maxminute := 55, [727].log_data[0].valid := 1, [727].log_data[1].valid := 1, [727].log_data[2].valid := 1, [727].log_data[3].valid := 1, [727].log_data[4].valid := 1, [727].log_data[5].valid := 1, [727].log_data[6].valid := 1, [727].log_data[7].valid := 1, [727].log_data[8].valid := 1, [727].log_data[9].valid := 1, [727].log_data[10].valid := 1, [727].log_data[11].valid := 1, [727].log_data[12].valid := 1, [727].log_data[13].valid := 1, [727].log_data[14].valid := 1, [727].log_data[15].valid := 1, [727].log_data[16].valid := 1, [727].log_data[17].valid := 1, [727].log_data[18].valid := 1, [727].log_data[19].valid := 1, [727].time.Year := 2023, [727].time.Month := 1, [727].time.Day := 12, [727].time.Hour := 4, [727].time.Minute := 59, [727].time.Second := 59, [728].log_data[0].min := 1.0, [728].log_data[0].max := 1.0, [728].log_data[0].total := 300.0, [728].log_data[0].time := 300.0, [728].log_data[0].valid := 1, [728].log_data[1].valid := 1, [728].log_data[2].valid := 1, [728].log_data[3].valid := 1, [728].log_data[4].valid := 1, [728].log_data[5].valid := 1, [728].log_data[6].valid := 1, [728].log_data[7].valid := 1, [728].log_data[8].valid := 1, [728].log_data[9].valid := 1, [728].log_data[10].valid := 1, [728].log_data[11].valid := 1, [728].log_data[12].valid := 1, [728].log_data[13].valid := 1, [728].log_data[14].valid := 1, [728].log_data[15].valid := 1, [728].log_data[16].valid := 1, [728].log_data[17].valid := 1,
        [728].log_data[18].valid := 1, [728].log_data[19].valid := 1, [728].time.Year := 2023, [728].time.Month := 1, [728].time.Day := 12, [728].time.Hour := 5, [728].time.Minute := 4, [728].time.Second := 59, [729].log_data[0].min := 1.0, [729].log_data[0].max := 1.0, [729].log_data[0].total := 300.0, [729].log_data[0].time := 300.0, [729].log_data[0].minminute := 5, [729].log_data[0].maxminute := 5, [729].log_data[0].valid := 1, [729].log_data[1].valid := 1, [729].log_data[2].valid := 1, [729].log_data[3].valid := 1, [729].log_data[4].valid := 1, [729].log_data[5].valid := 1, [729].log_data[6].valid := 1, [729].log_data[7].valid := 1, [729].log_data[8].valid := 1, [729].log_data[9].valid := 1, [729].log_data[10].valid := 1, [729].log_data[11].valid := 1, [729].log_data[12].valid := 1, [729].log_data[13].valid := 1, [729].log_data[14].valid := 1, [729].log_data[15].valid := 1, [729].log_data[16].valid := 1, [729].log_data[17].valid := 1, [729].log_data[18].valid := 1, [729].log_data[19].valid := 1, [729].time.Year := 2023, [729].time.Month := 1, [729].time.Day := 12, [729].time.Hour := 5, [729].time.Minute := 9, [729].time.Second := 59, [730].log_data[0].min := 1.0, [730].log_data[0].max := 1.0, [730].log_data[0].total := 300.0, [730].log_data[0].time := 300.0, [730].log_data[0].minminute := 10, [730].log_data[0].maxminute := 10, [730].log_data[0].valid := 1, [730].log_data[1].valid := 1, [730].log_data[2].valid := 1, [730].log_data[3].valid := 1, [730].log_data[4].valid := 1, [730].log_data[5].valid := 1, [730].log_data[6].valid := 1, [730].log_data[7].valid := 1, [730].log_data[8].valid := 1, [730].log_data[9].valid := 1, [730].log_data[10].valid := 1, [730].log_data[11].valid := 1, [730].log_data[12].valid := 1, [730].log_data[13].valid := 1,
        [730].log_data[14].valid := 1, [730].log_data[15].valid := 1, [730].log_data[16].valid := 1, [730].log_data[17].valid := 1, [730].log_data[18].valid := 1, [730].log_data[19].valid := 1, [730].time.Year := 2023, [730].time.Month := 1, [730].time.Day := 12, [730].time.Hour := 5, [730].time.Minute := 14, [730].time.Second := 59, [731].log_data[0].min := 1.0, [731].log_data[0].max := 1.0, [731].log_data[0].total := 300.0, [731].log_data[0].time := 300.0, [731].log_data[0].minminute := 15, [731].log_data[0].maxminute := 15, [731].log_data[0].valid := 1, [731].log_data[1].valid := 1, [731].log_data[2].valid := 1, [731].log_data[3].valid := 1, [731].log_data[4].valid := 1, [731].log_data[5].valid := 1, [731].log_data[6].valid := 1, [731].log_data[7].valid := 1, [731].log_data[8].valid := 1, [731].log_data[9].valid := 1, [731].log_data[10].valid := 1, [731].log_data[11].valid := 1, [731].log_data[12].valid := 1, [731].log_data[13].valid := 1, [731].log_data[14].valid := 1, [731].log_data[15].valid := 1, [731].log_data[16].valid := 1, [731].log_data[17].valid := 1, [731].log_data[18].valid := 1, [731].log_data[19].valid := 1, [731].time.Year := 2023, [731].time.Month := 1, [731].time.Day := 12, [731].time.Hour := 5, [731].time.Minute := 19, [731].time.Second := 59, [732].log_data[0].min := 1.0, [732].log_data[0].max := 1.0, [732].log_data[0].total := 300.0, [732].log_data[0].time := 300.0, [732].log_data[0].minminute := 20, [732].log_data[0].maxminute := 20, [732].log_data[0].valid := 1, [732].log_data[1].valid := 1, [732].log_data[2].valid := 1, [732].log_data[3].valid := 1, [732].log_data[4].valid := 1, [732].log_data[5].valid := 1, [732].log_data[6].valid := 1, [732].log_data[7].valid := 1, [732].log_data[8].valid := 1, [732].log_data[9].valid := 1,
        [732].log_data[10].valid := 1, [732].log_data[11].valid := 1, [732].log_data[12].valid := 1, [732].log_data[13].valid := 1, [732].log_data[14].valid := 1, [732].log_data[15].valid := 1, [732].log_data[16].valid := 1, [732].log_data[17].valid := 1, [732].log_data[18].valid := 1, [732].log_data[19].valid := 1, [732].time.Year := 2023, [732].time.Month := 1, [732].time.Day := 12, [732].time.Hour := 5, [732].time.Minute := 24, [732].time.Second := 59, [733].log_data[0].min := 1.0, [733].log_data[0].max := 1.0, [733].log_data[0].total := 300.0, [733].log_data[0].time := 300.0, [733].log_data[0].minminute := 25, [733].log_data[0].maxminute := 25, [733].log_data[0].valid := 1, [733].log_data[1].valid := 1, [733].log_data[2].valid := 1, [733].log_data[3].valid := 1, [733].log_data[4].valid := 1, [733].log_data[5].valid := 1, [733].log_data[6].valid := 1, [733].log_data[7].valid := 1, [733].log_data[8].valid := 1, [733].log_data[9].valid := 1, [733].log_data[10].valid := 1, [733].log_data[11].valid := 1, [733].log_data[12].valid := 1, [733].log_data[13].valid := 1, [733].log_data[14].valid := 1, [733].log_data[15].valid := 1, [733].log_data[16].valid := 1, [733].log_data[17].valid := 1, [733].log_data[18].valid := 1, [733].log_data[19].valid := 1, [733].time.Year := 2023, [733].time.Month := 1, [733].time.Day := 12, [733].time.Hour := 5, [733].time.Minute := 29, [733].time.Second := 59, [734].log_data[0].min := 1.0, [734].log_data[0].max := 1.0, [734].log_data[0].total := 300.0, [734].log_data[0].time := 300.0, [734].log_data[0].minminute := 30, [734].log_data[0].maxminute := 30, [734].log_data[0].valid := 1, [734].log_data[1].valid := 1, [734].log_data[2].valid := 1, [734].log_data[3].valid := 1, [734].log_data[4].valid := 1, [734].log_data[5].valid := 1,
        [734].log_data[6].valid := 1, [734].log_data[7].valid := 1, [734].log_data[8].valid := 1, [734].log_data[9].valid := 1, [734].log_data[10].valid := 1, [734].log_data[11].valid := 1, [734].log_data[12].valid := 1, [734].log_data[13].valid := 1, [734].log_data[14].valid := 1, [734].log_data[15].valid := 1, [734].log_data[16].valid := 1, [734].log_data[17].valid := 1, [734].log_data[18].valid := 1, [734].log_data[19].valid := 1, [734].time.Year := 2023, [734].time.Month := 1, [734].time.Day := 12, [734].time.Hour := 5, [734].time.Minute := 34, [734].time.Second := 59, [735].log_data[0].min := 1.0, [735].log_data[0].max := 1.0, [735].log_data[0].total := 300.0, [735].log_data[0].time := 300.0, [735].log_data[0].minminute := 35, [735].log_data[0].maxminute := 35, [735].log_data[0].valid := 1, [735].log_data[1].valid := 1, [735].log_data[2].valid := 1, [735].log_data[3].valid := 1, [735].log_data[4].valid := 1, [735].log_data[5].valid := 1, [735].log_data[6].valid := 1, [735].log_data[7].valid := 1, [735].log_data[8].valid := 1, [735].log_data[9].valid := 1, [735].log_data[10].valid := 1, [735].log_data[11].valid := 1, [735].log_data[12].valid := 1, [735].log_data[13].valid := 1, [735].log_data[14].valid := 1, [735].log_data[15].valid := 1, [735].log_data[16].valid := 1, [735].log_data[17].valid := 1, [735].log_data[18].valid := 1, [735].log_data[19].valid := 1, [735].time.Year := 2023, [735].time.Month := 1, [735].time.Day := 12, [735].time.Hour := 5, [735].time.Minute := 39, [735].time.Second := 59, [736].log_data[0].min := 1.0, [736].log_data[0].max := 1.0, [736].log_data[0].total := 300.0, [736].log_data[0].time := 300.0, [736].log_data[0].minminute := 40, [736].log_data[0].maxminute := 40, [736].log_data[0].valid := 1, [736].log_data[1].valid := 1,
        [736].log_data[2].valid := 1, [736].log_data[3].valid := 1, [736].log_data[4].valid := 1, [736].log_data[5].valid := 1, [736].log_data[6].valid := 1, [736].log_data[7].valid := 1, [736].log_data[8].valid := 1, [736].log_data[9].valid := 1, [736].log_data[10].valid := 1, [736].log_data[11].valid := 1, [736].log_data[12].valid := 1, [736].log_data[13].valid := 1, [736].log_data[14].valid := 1, [736].log_data[15].valid := 1, [736].log_data[16].valid := 1, [736].log_data[17].valid := 1, [736].log_data[18].valid := 1, [736].log_data[19].valid := 1, [736].time.Year := 2023, [736].time.Month := 1, [736].time.Day := 12, [736].time.Hour := 5, [736].time.Minute := 44, [736].time.Second := 59, [737].log_data[0].min := 1.0, [737].log_data[0].max := 1.0, [737].log_data[0].total := 300.0, [737].log_data[0].time := 300.0, [737].log_data[0].minminute := 45, [737].log_data[0].maxminute := 45, [737].log_data[0].valid := 1, [737].log_data[1].valid := 1, [737].log_data[2].valid := 1, [737].log_data[3].valid := 1, [737].log_data[4].valid := 1, [737].log_data[5].valid := 1, [737].log_data[6].valid := 1, [737].log_data[7].valid := 1, [737].log_data[8].valid := 1, [737].log_data[9].valid := 1, [737].log_data[10].valid := 1, [737].log_data[11].valid := 1, [737].log_data[12].valid := 1, [737].log_data[13].valid := 1, [737].log_data[14].valid := 1, [737].log_data[15].valid := 1, [737].log_data[16].valid := 1, [737].log_data[17].valid := 1, [737].log_data[18].valid := 1, [737].log_data[19].valid := 1, [737].time.Year := 2023, [737].time.Month := 1, [737].time.Day := 12, [737].time.Hour := 5, [737].time.Minute := 49, [737].time.Second := 59, [738].log_data[0].min := 1.0, [738].log_data[0].max := 1.0, [738].log_data[0].total := 300.0, [738].log_data[0].time := 300.0,
        [738].log_data[0].minminute := 50, [738].log_data[0].maxminute := 50, [738].log_data[0].valid := 1, [738].log_data[1].valid := 1, [738].log_data[2].valid := 1, [738].log_data[3].valid := 1, [738].log_data[4].valid := 1, [738].log_data[5].valid := 1, [738].log_data[6].valid := 1, [738].log_data[7].valid := 1, [738].log_data[8].valid := 1, [738].log_data[9].valid := 1, [738].log_data[10].valid := 1, [738].log_data[11].valid := 1, [738].log_data[12].valid := 1, [738].log_data[13].valid := 1, [738].log_data[14].valid := 1, [738].log_data[15].valid := 1, [738].log_data[16].valid := 1, [738].log_data[17].valid := 1, [738].log_data[18].valid := 1, [738].log_data[19].valid := 1, [738].time.Year := 2023, [738].time.Month := 1, [738].time.Day := 12, [738].time.Hour := 5, [738].time.Minute := 54, [738].time.Second := 59, [739].log_data[0].min := 1.0, [739].log_data[0].max := 1.0, [739].log_data[0].total := 300.0, [739].log_data[0].time := 300.0, [739].log_data[0].minminute := 55, [739].log_data[0].maxminute := 55, [739].log_data[0].valid := 1, [739].log_data[1].valid := 1, [739].log_data[2].valid := 1, [739].log_data[3].valid := 1, [739].log_data[4].valid := 1, [739].log_data[5].valid := 1, [739].log_data[6].valid := 1, [739].log_data[7].valid := 1, [739].log_data[8].valid := 1, [739].log_data[9].valid := 1, [739].log_data[10].valid := 1, [739].log_data[11].valid := 1, [739].log_data[12].valid := 1, [739].log_data[13].valid := 1, [739].log_data[14].valid := 1, [739].log_data[15].valid := 1, [739].log_data[16].valid := 1, [739].log_data[17].valid := 1, [739].log_data[18].valid := 1, [739].log_data[19].valid := 1, [739].time.Year := 2023, [739].time.Month := 1, [739].time.Day := 12, [739].time.Hour := 5, [739].time.Minute := 59, [739].time.Second := 59,
        [740].log_data[0].min := 1.0, [740].log_data[0].max := 1.0, [740].log_data[0].total := 300.0, [740].log_data[0].time := 300.0, [740].log_data[0].valid := 1, [740].log_data[1].valid := 1, [740].log_data[2].valid := 1, [740].log_data[3].valid := 1, [740].log_data[4].valid := 1, [740].log_data[5].valid := 1, [740].log_data[6].valid := 1, [740].log_data[7].valid := 1, [740].log_data[8].valid := 1, [740].log_data[9].valid := 1, [740].log_data[10].valid := 1, [740].log_data[11].valid := 1, [740].log_data[12].valid := 1, [740].log_data[13].valid := 1, [740].log_data[14].valid := 1, [740].log_data[15].valid := 1, [740].log_data[16].valid := 1, [740].log_data[17].valid := 1, [740].log_data[18].valid := 1, [740].log_data[19].valid := 1, [740].time.Year := 2023, [740].time.Month := 1, [740].time.Day := 12, [740].time.Hour := 6, [740].time.Minute := 4, [740].time.Second := 59, [741].log_data[0].min := 1.0, [741].log_data[0].max := 1.0, [741].log_data[0].total := 300.0, [741].log_data[0].time := 300.0, [741].log_data[0].minminute := 5, [741].log_data[0].maxminute := 5, [741].log_data[0].valid := 1, [741].log_data[1].valid := 1, [741].log_data[2].valid := 1, [741].log_data[3].valid := 1, [741].log_data[4].valid := 1, [741].log_data[5].valid := 1, [741].log_data[6].valid := 1, [741].log_data[7].valid := 1, [741].log_data[8].valid := 1, [741].log_data[9].valid := 1, [741].log_data[10].valid := 1, [741].log_data[11].valid := 1, [741].log_data[12].valid := 1, [741].log_data[13].valid := 1, [741].log_data[14].valid := 1, [741].log_data[15].valid := 1, [741].log_data[16].valid := 1, [741].log_data[17].valid := 1, [741].log_data[18].valid := 1, [741].log_data[19].valid := 1, [741].time.Year := 2023, [741].time.Month := 1, [741].time.Day := 12, [741].time.Hour := 6,
        [741].time.Minute := 9, [741].time.Second := 59, [742].log_data[0].min := 1.0, [742].log_data[0].max := 1.0, [742].log_data[0].total := 300.0, [742].log_data[0].time := 300.0, [742].log_data[0].minminute := 10, [742].log_data[0].maxminute := 10, [742].log_data[0].valid := 1, [742].log_data[1].valid := 1, [742].log_data[2].valid := 1, [742].log_data[3].valid := 1, [742].log_data[4].valid := 1, [742].log_data[5].valid := 1, [742].log_data[6].valid := 1, [742].log_data[7].valid := 1, [742].log_data[8].valid := 1, [742].log_data[9].valid := 1, [742].log_data[10].valid := 1, [742].log_data[11].valid := 1, [742].log_data[12].valid := 1, [742].log_data[13].valid := 1, [742].log_data[14].valid := 1, [742].log_data[15].valid := 1, [742].log_data[16].valid := 1, [742].log_data[17].valid := 1, [742].log_data[18].valid := 1, [742].log_data[19].valid := 1, [742].time.Year := 2023, [742].time.Month := 1, [742].time.Day := 12, [742].time.Hour := 6, [742].time.Minute := 14, [742].time.Second := 59, [743].log_data[0].min := 1.0, [743].log_data[0].max := 1.0, [743].log_data[0].total := 300.0, [743].log_data[0].time := 300.0, [743].log_data[0].minminute := 15, [743].log_data[0].maxminute := 15, [743].log_data[0].valid := 1, [743].log_data[1].valid := 1, [743].log_data[2].valid := 1, [743].log_data[3].valid := 1, [743].log_data[4].valid := 1, [743].log_data[5].valid := 1, [743].log_data[6].valid := 1, [743].log_data[7].valid := 1, [743].log_data[8].valid := 1, [743].log_data[9].valid := 1, [743].log_data[10].valid := 1, [743].log_data[11].valid := 1, [743].log_data[12].valid := 1, [743].log_data[13].valid := 1, [743].log_data[14].valid := 1, [743].log_data[15].valid := 1, [743].log_data[16].valid := 1, [743].log_data[17].valid := 1, [743].log_data[18].valid := 1, [743].log_data[19].valid := 1,
        [743].time.Year := 2023, [743].time.Month := 1, [743].time.Day := 12, [743].time.Hour := 6, [743].time.Minute := 19, [743].time.Second := 59, [744].log_data[0].min := 1.0, [744].log_data[0].max := 1.0, [744].log_data[0].total := 300.0, [744].log_data[0].time := 300.0, [744].log_data[0].minminute := 20, [744].log_data[0].maxminute := 20, [744].log_data[0].valid := 1, [744].log_data[1].valid := 1, [744].log_data[2].valid := 1, [744].log_data[3].valid := 1, [744].log_data[4].valid := 1, [744].log_data[5].valid := 1, [744].log_data[6].valid := 1, [744].log_data[7].valid := 1, [744].log_data[8].valid := 1, [744].log_data[9].valid := 1, [744].log_data[10].valid := 1, [744].log_data[11].valid := 1, [744].log_data[12].valid := 1, [744].log_data[13].valid := 1, [744].log_data[14].valid := 1, [744].log_data[15].valid := 1, [744].log_data[16].valid := 1, [744].log_data[17].valid := 1, [744].log_data[18].valid := 1, [744].log_data[19].valid := 1, [744].time.Year := 2023, [744].time.Month := 1, [744].time.Day := 12, [744].time.Hour := 6, [744].time.Minute := 24, [744].time.Second := 59, [745].log_data[0].min := 1.0, [745].log_data[0].max := 1.0, [745].log_data[0].total := 300.0, [745].log_data[0].time := 300.0, [745].log_data[0].minminute := 25, [745].log_data[0].maxminute := 25, [745].log_data[0].valid := 1, [745].log_data[1].valid := 1, [745].log_data[2].valid := 1, [745].log_data[3].valid := 1, [745].log_data[4].valid := 1, [745].log_data[5].valid := 1, [745].log_data[6].valid := 1, [745].log_data[7].valid := 1, [745].log_data[8].valid := 1, [745].log_data[9].valid := 1, [745].log_data[10].valid := 1, [745].log_data[11].valid := 1, [745].log_data[12].valid := 1, [745].log_data[13].valid := 1, [745].log_data[14].valid := 1, [745].log_data[15].valid := 1,
        [745].log_data[16].valid := 1, [745].log_data[17].valid := 1, [745].log_data[18].valid := 1, [745].log_data[19].valid := 1, [745].time.Year := 2023, [745].time.Month := 1, [745].time.Day := 12, [745].time.Hour := 6, [745].time.Minute := 29, [745].time.Second := 59, [746].log_data[0].min := 1.0, [746].log_data[0].max := 1.0, [746].log_data[0].total := 300.0, [746].log_data[0].time := 300.0, [746].log_data[0].minminute := 30, [746].log_data[0].maxminute := 30, [746].log_data[0].valid := 1, [746].log_data[1].valid := 1, [746].log_data[2].valid := 1, [746].log_data[3].valid := 1, [746].log_data[4].valid := 1, [746].log_data[5].valid := 1, [746].log_data[6].valid := 1, [746].log_data[7].valid := 1, [746].log_data[8].valid := 1, [746].log_data[9].valid := 1, [746].log_data[10].valid := 1, [746].log_data[11].valid := 1, [746].log_data[12].valid := 1, [746].log_data[13].valid := 1, [746].log_data[14].valid := 1, [746].log_data[15].valid := 1, [746].log_data[16].valid := 1, [746].log_data[17].valid := 1, [746].log_data[18].valid := 1, [746].log_data[19].valid := 1, [746].time.Year := 2023, [746].time.Month := 1, [746].time.Day := 12, [746].time.Hour := 6, [746].time.Minute := 34, [746].time.Second := 59, [747].log_data[0].min := 1.0, [747].log_data[0].max := 1.0, [747].log_data[0].total := 300.0, [747].log_data[0].time := 300.0, [747].log_data[0].minminute := 35, [747].log_data[0].maxminute := 35, [747].log_data[0].valid := 1, [747].log_data[1].valid := 1, [747].log_data[2].valid := 1, [747].log_data[3].valid := 1, [747].log_data[4].valid := 1, [747].log_data[5].valid := 1, [747].log_data[6].valid := 1, [747].log_data[7].valid := 1, [747].log_data[8].valid := 1, [747].log_data[9].valid := 1, [747].log_data[10].valid := 1, [747].log_data[11].valid := 1,
        [747].log_data[12].valid := 1, [747].log_data[13].valid := 1, [747].log_data[14].valid := 1, [747].log_data[15].valid := 1, [747].log_data[16].valid := 1, [747].log_data[17].valid := 1, [747].log_data[18].valid := 1, [747].log_data[19].valid := 1, [747].time.Year := 2023, [747].time.Month := 1, [747].time.Day := 12, [747].time.Hour := 6, [747].time.Minute := 39, [747].time.Second := 59, [748].log_data[0].min := 1.0, [748].log_data[0].max := 1.0, [748].log_data[0].total := 300.0, [748].log_data[0].time := 300.0, [748].log_data[0].minminute := 40, [748].log_data[0].maxminute := 40, [748].log_data[0].valid := 1, [748].log_data[1].valid := 1, [748].log_data[2].valid := 1, [748].log_data[3].valid := 1, [748].log_data[4].valid := 1, [748].log_data[5].valid := 1, [748].log_data[6].valid := 1, [748].log_data[7].valid := 1, [748].log_data[8].valid := 1, [748].log_data[9].valid := 1, [748].log_data[10].valid := 1, [748].log_data[11].valid := 1, [748].log_data[12].valid := 1, [748].log_data[13].valid := 1, [748].log_data[14].valid := 1, [748].log_data[15].valid := 1, [748].log_data[16].valid := 1, [748].log_data[17].valid := 1, [748].log_data[18].valid := 1, [748].log_data[19].valid := 1, [748].time.Year := 2023, [748].time.Month := 1, [748].time.Day := 12, [748].time.Hour := 6, [748].time.Minute := 44, [748].time.Second := 59, [749].log_data[0].min := 1.0, [749].log_data[0].max := 1.0, [749].log_data[0].total := 300.0, [749].log_data[0].time := 300.0, [749].log_data[0].minminute := 45, [749].log_data[0].maxminute := 45, [749].log_data[0].valid := 1, [749].log_data[1].valid := 1, [749].log_data[2].valid := 1, [749].log_data[3].valid := 1, [749].log_data[4].valid := 1, [749].log_data[5].valid := 1, [749].log_data[6].valid := 1, [749].log_data[7].valid := 1,
        [749].log_data[8].valid := 1, [749].log_data[9].valid := 1, [749].log_data[10].valid := 1, [749].log_data[11].valid := 1, [749].log_data[12].valid := 1, [749].log_data[13].valid := 1, [749].log_data[14].valid := 1, [749].log_data[15].valid := 1, [749].log_data[16].valid := 1, [749].log_data[17].valid := 1, [749].log_data[18].valid := 1, [749].log_data[19].valid := 1, [749].time.Year := 2023, [749].time.Month := 1, [749].time.Day := 12, [749].time.Hour := 6, [749].time.Minute := 49, [749].time.Second := 59, [750].log_data[0].min := 1.0, [750].log_data[0].max := 1.0, [750].log_data[0].total := 300.0, [750].log_data[0].time := 300.0, [750].log_data[0].minminute := 50, [750].log_data[0].maxminute := 50, [750].log_data[0].valid := 1, [750].log_data[1].valid := 1, [750].log_data[2].valid := 1, [750].log_data[3].valid := 1, [750].log_data[4].valid := 1, [750].log_data[5].valid := 1, [750].log_data[6].valid := 1, [750].log_data[7].valid := 1, [750].log_data[8].valid := 1, [750].log_data[9].valid := 1, [750].log_data[10].valid := 1, [750].log_data[11].valid := 1, [750].log_data[12].valid := 1, [750].log_data[13].valid := 1, [750].log_data[14].valid := 1, [750].log_data[15].valid := 1, [750].log_data[16].valid := 1, [750].log_data[17].valid := 1, [750].log_data[18].valid := 1, [750].log_data[19].valid := 1, [750].time.Year := 2023, [750].time.Month := 1, [750].time.Day := 12, [750].time.Hour := 6, [750].time.Minute := 54, [750].time.Second := 59, [751].log_data[0].min := 1.0, [751].log_data[0].max := 1.0, [751].log_data[0].total := 300.0, [751].log_data[0].time := 300.0, [751].log_data[0].minminute := 55, [751].log_data[0].maxminute := 55, [751].log_data[0].valid := 1, [751].log_data[1].valid := 1, [751].log_data[2].valid := 1, [751].log_data[3].valid := 1,
        [751].log_data[4].valid := 1, [751].log_data[5].valid := 1, [751].log_data[6].valid := 1, [751].log_data[7].valid := 1, [751].log_data[8].valid := 1, [751].log_data[9].valid := 1, [751].log_data[10].valid := 1, [751].log_data[11].valid := 1, [751].log_data[12].valid := 1, [751].log_data[13].valid := 1, [751].log_data[14].valid := 1, [751].log_data[15].valid := 1, [751].log_data[16].valid := 1, [751].log_data[17].valid := 1, [751].log_data[18].valid := 1, [751].log_data[19].valid := 1, [751].time.Year := 2023, [751].time.Month := 1, [751].time.Day := 12, [751].time.Hour := 6, [751].time.Minute := 59, [751].time.Second := 59, [752].log_data[0].min := 1.0, [752].log_data[0].max := 1.0, [752].log_data[0].total := 300.0, [752].log_data[0].time := 300.0, [752].log_data[0].valid := 1, [752].log_data[1].valid := 1, [752].log_data[2].valid := 1, [752].log_data[3].valid := 1, [752].log_data[4].valid := 1, [752].log_data[5].valid := 1, [752].log_data[6].valid := 1, [752].log_data[7].valid := 1, [752].log_data[8].valid := 1, [752].log_data[9].valid := 1, [752].log_data[10].valid := 1, [752].log_data[11].valid := 1, [752].log_data[12].valid := 1, [752].log_data[13].valid := 1, [752].log_data[14].valid := 1, [752].log_data[15].valid := 1, [752].log_data[16].valid := 1, [752].log_data[17].valid := 1, [752].log_data[18].valid := 1, [752].log_data[19].valid := 1, [752].time.Year := 2023, [752].time.Month := 1, [752].time.Day := 12, [752].time.Hour := 7, [752].time.Minute := 4, [752].time.Second := 59, [753].log_data[0].min := 1.0, [753].log_data[0].max := 1.0, [753].log_data[0].total := 300.0, [753].log_data[0].time := 300.0, [753].log_data[0].minminute := 5, [753].log_data[0].maxminute := 5, [753].log_data[0].valid := 1, [753].log_data[1].valid := 1,
        [753].log_data[2].valid := 1, [753].log_data[3].valid := 1, [753].log_data[4].valid := 1, [753].log_data[5].valid := 1, [753].log_data[6].valid := 1, [753].log_data[7].valid := 1, [753].log_data[8].valid := 1, [753].log_data[9].valid := 1, [753].log_data[10].valid := 1, [753].log_data[11].valid := 1, [753].log_data[12].valid := 1, [753].log_data[13].valid := 1, [753].log_data[14].valid := 1, [753].log_data[15].valid := 1, [753].log_data[16].valid := 1, [753].log_data[17].valid := 1, [753].log_data[18].valid := 1, [753].log_data[19].valid := 1, [753].time.Year := 2023, [753].time.Month := 1, [753].time.Day := 12, [753].time.Hour := 7, [753].time.Minute := 9, [753].time.Second := 59, [754].log_data[0].min := 1.0, [754].log_data[0].max := 1.0, [754].log_data[0].total := 300.0, [754].log_data[0].time := 300.0, [754].log_data[0].minminute := 10, [754].log_data[0].maxminute := 10, [754].log_data[0].valid := 1, [754].log_data[1].valid := 1, [754].log_data[2].valid := 1, [754].log_data[3].valid := 1, [754].log_data[4].valid := 1, [754].log_data[5].valid := 1, [754].log_data[6].valid := 1, [754].log_data[7].valid := 1, [754].log_data[8].valid := 1, [754].log_data[9].valid := 1, [754].log_data[10].valid := 1, [754].log_data[11].valid := 1, [754].log_data[12].valid := 1, [754].log_data[13].valid := 1, [754].log_data[14].valid := 1, [754].log_data[15].valid := 1, [754].log_data[16].valid := 1, [754].log_data[17].valid := 1, [754].log_data[18].valid := 1, [754].log_data[19].valid := 1, [754].time.Year := 2023, [754].time.Month := 1, [754].time.Day := 12, [754].time.Hour := 7, [754].time.Minute := 14, [754].time.Second := 59, [755].log_data[0].min := 1.0, [755].log_data[0].max := 1.0, [755].log_data[0].total := 300.0, [755].log_data[0].time := 300.0,
        [755].log_data[0].minminute := 15, [755].log_data[0].maxminute := 15, [755].log_data[0].valid := 1, [755].log_data[1].valid := 1, [755].log_data[2].valid := 1, [755].log_data[3].valid := 1, [755].log_data[4].valid := 1, [755].log_data[5].valid := 1, [755].log_data[6].valid := 1, [755].log_data[7].valid := 1, [755].log_data[8].valid := 1, [755].log_data[9].valid := 1, [755].log_data[10].valid := 1, [755].log_data[11].valid := 1, [755].log_data[12].valid := 1, [755].log_data[13].valid := 1, [755].log_data[14].valid := 1, [755].log_data[15].valid := 1, [755].log_data[16].valid := 1, [755].log_data[17].valid := 1, [755].log_data[18].valid := 1, [755].log_data[19].valid := 1, [755].time.Year := 2023, [755].time.Month := 1, [755].time.Day := 12, [755].time.Hour := 7, [755].time.Minute := 19, [755].time.Second := 59, [756].log_data[0].min := 1.0, [756].log_data[0].max := 1.0, [756].log_data[0].total := 300.0, [756].log_data[0].time := 300.0, [756].log_data[0].minminute := 20, [756].log_data[0].maxminute := 20, [756].log_data[0].valid := 1, [756].log_data[1].valid := 1, [756].log_data[2].valid := 1, [756].log_data[3].valid := 1, [756].log_data[4].valid := 1, [756].log_data[5].valid := 1, [756].log_data[6].valid := 1, [756].log_data[7].valid := 1, [756].log_data[8].valid := 1, [756].log_data[9].valid := 1, [756].log_data[10].valid := 1, [756].log_data[11].valid := 1, [756].log_data[12].valid := 1, [756].log_data[13].valid := 1, [756].log_data[14].valid := 1, [756].log_data[15].valid := 1, [756].log_data[16].valid := 1, [756].log_data[17].valid := 1, [756].log_data[18].valid := 1, [756].log_data[19].valid := 1, [756].time.Year := 2023, [756].time.Month := 1, [756].time.Day := 12, [756].time.Hour := 7, [756].time.Minute := 24, [756].time.Second := 59,
        [757].log_data[0].min := 1.0, [757].log_data[0].max := 1.0, [757].log_data[0].total := 300.0, [757].log_data[0].time := 300.0, [757].log_data[0].minminute := 25, [757].log_data[0].maxminute := 25, [757].log_data[0].valid := 1, [757].log_data[1].valid := 1, [757].log_data[2].valid := 1, [757].log_data[3].valid := 1, [757].log_data[4].valid := 1, [757].log_data[5].valid := 1, [757].log_data[6].valid := 1, [757].log_data[7].valid := 1, [757].log_data[8].valid := 1, [757].log_data[9].valid := 1, [757].log_data[10].valid := 1, [757].log_data[11].valid := 1, [757].log_data[12].valid := 1, [757].log_data[13].valid := 1, [757].log_data[14].valid := 1, [757].log_data[15].valid := 1, [757].log_data[16].valid := 1, [757].log_data[17].valid := 1, [757].log_data[18].valid := 1, [757].log_data[19].valid := 1, [757].time.Year := 2023, [757].time.Month := 1, [757].time.Day := 12, [757].time.Hour := 7, [757].time.Minute := 29, [757].time.Second := 59, [758].log_data[0].min := 1.0, [758].log_data[0].max := 1.0, [758].log_data[0].total := 300.0, [758].log_data[0].time := 300.0, [758].log_data[0].minminute := 30, [758].log_data[0].maxminute := 30, [758].log_data[0].valid := 1, [758].log_data[1].valid := 1, [758].log_data[2].valid := 1, [758].log_data[3].valid := 1, [758].log_data[4].valid := 1, [758].log_data[5].valid := 1, [758].log_data[6].valid := 1, [758].log_data[7].valid := 1, [758].log_data[8].valid := 1, [758].log_data[9].valid := 1, [758].log_data[10].valid := 1, [758].log_data[11].valid := 1, [758].log_data[12].valid := 1, [758].log_data[13].valid := 1, [758].log_data[14].valid := 1, [758].log_data[15].valid := 1, [758].log_data[16].valid := 1, [758].log_data[17].valid := 1, [758].log_data[18].valid := 1, [758].log_data[19].valid := 1, [758].time.Year := 2023, [758].time.Month := 1,
        [758].time.Day := 12, [758].time.Hour := 7, [758].time.Minute := 34, [758].time.Second := 59, [759].log_data[0].min := 1.0, [759].log_data[0].max := 1.0, [759].log_data[0].total := 300.0, [759].log_data[0].time := 300.0, [759].log_data[0].minminute := 35, [759].log_data[0].maxminute := 35, [759].log_data[0].valid := 1, [759].log_data[1].valid := 1, [759].log_data[2].valid := 1, [759].log_data[3].valid := 1, [759].log_data[4].valid := 1, [759].log_data[5].valid := 1, [759].log_data[6].valid := 1, [759].log_data[7].valid := 1, [759].log_data[8].valid := 1, [759].log_data[9].valid := 1, [759].log_data[10].valid := 1, [759].log_data[11].valid := 1, [759].log_data[12].valid := 1, [759].log_data[13].valid := 1, [759].log_data[14].valid := 1, [759].log_data[15].valid := 1, [759].log_data[16].valid := 1, [759].log_data[17].valid := 1, [759].log_data[18].valid := 1, [759].log_data[19].valid := 1, [759].time.Year := 2023, [759].time.Month := 1, [759].time.Day := 12, [759].time.Hour := 7, [759].time.Minute := 39, [759].time.Second := 59, [760].log_data[0].min := 1.0, [760].log_data[0].max := 1.0, [760].log_data[0].total := 300.0, [760].log_data[0].time := 300.0, [760].log_data[0].minminute := 40, [760].log_data[0].maxminute := 40, [760].log_data[0].valid := 1, [760].log_data[1].valid := 1, [760].log_data[2].valid := 1, [760].log_data[3].valid := 1, [760].log_data[4].valid := 1, [760].log_data[5].valid := 1, [760].log_data[6].valid := 1, [760].log_data[7].valid := 1, [760].log_data[8].valid := 1, [760].log_data[9].valid := 1, [760].log_data[10].valid := 1, [760].log_data[11].valid := 1, [760].log_data[12].valid := 1, [760].log_data[13].valid := 1, [760].log_data[14].valid := 1, [760].log_data[15].valid := 1, [760].log_data[16].valid := 1, [760].log_data[17].valid := 1,
        [760].log_data[18].valid := 1, [760].log_data[19].valid := 1, [760].time.Year := 2023, [760].time.Month := 1, [760].time.Day := 12, [760].time.Hour := 7, [760].time.Minute := 44, [760].time.Second := 59, [761].log_data[0].min := 1.0, [761].log_data[0].max := 1.0, [761].log_data[0].total := 300.0, [761].log_data[0].time := 300.0, [761].log_data[0].minminute := 45, [761].log_data[0].maxminute := 45, [761].log_data[0].valid := 1, [761].log_data[1].valid := 1, [761].log_data[2].valid := 1, [761].log_data[3].valid := 1, [761].log_data[4].valid := 1, [761].log_data[5].valid := 1, [761].log_data[6].valid := 1, [761].log_data[7].valid := 1, [761].log_data[8].valid := 1, [761].log_data[9].valid := 1, [761].log_data[10].valid := 1, [761].log_data[11].valid := 1, [761].log_data[12].valid := 1, [761].log_data[13].valid := 1, [761].log_data[14].valid := 1, [761].log_data[15].valid := 1, [761].log_data[16].valid := 1, [761].log_data[17].valid := 1, [761].log_data[18].valid := 1, [761].log_data[19].valid := 1, [761].time.Year := 2023, [761].time.Month := 1, [761].time.Day := 12, [761].time.Hour := 7, [761].time.Minute := 49, [761].time.Second := 59, [762].log_data[0].min := 1.0, [762].log_data[0].max := 1.0, [762].log_data[0].total := 300.0, [762].log_data[0].time := 300.0, [762].log_data[0].minminute := 50, [762].log_data[0].maxminute := 50, [762].log_data[0].valid := 1, [762].log_data[1].valid := 1, [762].log_data[2].valid := 1, [762].log_data[3].valid := 1, [762].log_data[4].valid := 1, [762].log_data[5].valid := 1, [762].log_data[6].valid := 1, [762].log_data[7].valid := 1, [762].log_data[8].valid := 1, [762].log_data[9].valid := 1, [762].log_data[10].valid := 1, [762].log_data[11].valid := 1, [762].log_data[12].valid := 1, [762].log_data[13].valid := 1,
        [762].log_data[14].valid := 1, [762].log_data[15].valid := 1, [762].log_data[16].valid := 1, [762].log_data[17].valid := 1, [762].log_data[18].valid := 1, [762].log_data[19].valid := 1, [762].time.Year := 2023, [762].time.Month := 1, [762].time.Day := 12, [762].time.Hour := 7, [762].time.Minute := 54, [762].time.Second := 59, [763].log_data[0].min := 1.0, [763].log_data[0].max := 1.0, [763].log_data[0].total := 300.0, [763].log_data[0].time := 300.0, [763].log_data[0].minminute := 55, [763].log_data[0].maxminute := 55, [763].log_data[0].valid := 1, [763].log_data[1].valid := 1, [763].log_data[2].valid := 1, [763].log_data[3].valid := 1, [763].log_data[4].valid := 1, [763].log_data[5].valid := 1, [763].log_data[6].valid := 1, [763].log_data[7].valid := 1, [763].log_data[8].valid := 1, [763].log_data[9].valid := 1, [763].log_data[10].valid := 1, [763].log_data[11].valid := 1, [763].log_data[12].valid := 1, [763].log_data[13].valid := 1, [763].log_data[14].valid := 1, [763].log_data[15].valid := 1, [763].log_data[16].valid := 1, [763].log_data[17].valid := 1, [763].log_data[18].valid := 1, [763].log_data[19].valid := 1, [763].time.Year := 2023, [763].time.Month := 1, [763].time.Day := 12, [763].time.Hour := 7, [763].time.Minute := 59, [763].time.Second := 59, [764].log_data[0].min := 1.0, [764].log_data[0].max := 1.0, [764].log_data[0].total := 300.0, [764].log_data[0].time := 300.0, [764].log_data[0].valid := 1, [764].log_data[1].valid := 1, [764].log_data[2].valid := 1, [764].log_data[3].valid := 1, [764].log_data[4].valid := 1, [764].log_data[5].valid := 1, [764].log_data[6].valid := 1, [764].log_data[7].valid := 1, [764].log_data[8].valid := 1, [764].log_data[9].valid := 1, [764].log_data[10].valid := 1, [764].log_data[11].valid := 1,
        [764].log_data[12].valid := 1, [764].log_data[13].valid := 1, [764].log_data[14].valid := 1, [764].log_data[15].valid := 1, [764].log_data[16].valid := 1, [764].log_data[17].valid := 1, [764].log_data[18].valid := 1, [764].log_data[19].valid := 1, [764].time.Year := 2023, [764].time.Month := 1, [764].time.Day := 12, [764].time.Hour := 8, [764].time.Minute := 4, [764].time.Second := 59, [765].log_data[0].min := 1.0, [765].log_data[0].max := 1.0, [765].log_data[0].total := 300.0, [765].log_data[0].time := 300.0, [765].log_data[0].minminute := 5, [765].log_data[0].maxminute := 5, [765].log_data[0].valid := 1, [765].log_data[1].valid := 1, [765].log_data[2].valid := 1, [765].log_data[3].valid := 1, [765].log_data[4].valid := 1, [765].log_data[5].valid := 1, [765].log_data[6].valid := 1, [765].log_data[7].valid := 1, [765].log_data[8].valid := 1, [765].log_data[9].valid := 1, [765].log_data[10].valid := 1, [765].log_data[11].valid := 1, [765].log_data[12].valid := 1, [765].log_data[13].valid := 1, [765].log_data[14].valid := 1, [765].log_data[15].valid := 1, [765].log_data[16].valid := 1, [765].log_data[17].valid := 1, [765].log_data[18].valid := 1, [765].log_data[19].valid := 1, [765].time.Year := 2023, [765].time.Month := 1, [765].time.Day := 12, [765].time.Hour := 8, [765].time.Minute := 9, [765].time.Second := 59, [766].log_data[0].min := 1.0, [766].log_data[0].max := 1.0, [766].log_data[0].total := 300.0, [766].log_data[0].time := 300.0, [766].log_data[0].minminute := 10, [766].log_data[0].maxminute := 10, [766].log_data[0].valid := 1, [766].log_data[1].valid := 1, [766].log_data[2].valid := 1, [766].log_data[3].valid := 1, [766].log_data[4].valid := 1, [766].log_data[5].valid := 1, [766].log_data[6].valid := 1, [766].log_data[7].valid := 1,
        [766].log_data[8].valid := 1, [766].log_data[9].valid := 1, [766].log_data[10].valid := 1, [766].log_data[11].valid := 1, [766].log_data[12].valid := 1, [766].log_data[13].valid := 1, [766].log_data[14].valid := 1, [766].log_data[15].valid := 1, [766].log_data[16].valid := 1, [766].log_data[17].valid := 1, [766].log_data[18].valid := 1, [766].log_data[19].valid := 1, [766].time.Year := 2023, [766].time.Month := 1, [766].time.Day := 12, [766].time.Hour := 8, [766].time.Minute := 14, [766].time.Second := 59, [767].log_data[0].min := 1.0, [767].log_data[0].max := 1.0, [767].log_data[0].total := 300.0, [767].log_data[0].time := 300.0, [767].log_data[0].minminute := 15, [767].log_data[0].maxminute := 15, [767].log_data[0].valid := 1, [767].log_data[1].valid := 1, [767].log_data[2].valid := 1, [767].log_data[3].valid := 1, [767].log_data[4].valid := 1, [767].log_data[5].valid := 1, [767].log_data[6].valid := 1, [767].log_data[7].valid := 1, [767].log_data[8].valid := 1, [767].log_data[9].valid := 1, [767].log_data[10].valid := 1, [767].log_data[11].valid := 1, [767].log_data[12].valid := 1, [767].log_data[13].valid := 1, [767].log_data[14].valid := 1, [767].log_data[15].valid := 1, [767].log_data[16].valid := 1, [767].log_data[17].valid := 1, [767].log_data[18].valid := 1, [767].log_data[19].valid := 1, [767].time.Year := 2023, [767].time.Month := 1, [767].time.Day := 12, [767].time.Hour := 8, [767].time.Minute := 19, [767].time.Second := 59, [768].log_data[0].min := 1.0, [768].log_data[0].max := 1.0, [768].log_data[0].total := 300.0, [768].log_data[0].time := 300.0, [768].log_data[0].minminute := 20, [768].log_data[0].maxminute := 20, [768].log_data[0].valid := 1, [768].log_data[1].valid := 1, [768].log_data[2].valid := 1, [768].log_data[3].valid := 1,
        [768].log_data[4].valid := 1, [768].log_data[5].valid := 1, [768].log_data[6].valid := 1, [768].log_data[7].valid := 1, [768].log_data[8].valid := 1, [768].log_data[9].valid := 1, [768].log_data[10].valid := 1, [768].log_data[11].valid := 1, [768].log_data[12].valid := 1, [768].log_data[13].valid := 1, [768].log_data[14].valid := 1, [768].log_data[15].valid := 1, [768].log_data[16].valid := 1, [768].log_data[17].valid := 1, [768].log_data[18].valid := 1, [768].log_data[19].valid := 1, [768].time.Year := 2023, [768].time.Month := 1, [768].time.Day := 12, [768].time.Hour := 8, [768].time.Minute := 24, [768].time.Second := 59, [769].log_data[0].min := 1.0, [769].log_data[0].max := 1.0, [769].log_data[0].total := 300.0, [769].log_data[0].time := 300.0, [769].log_data[0].minminute := 25, [769].log_data[0].maxminute := 25, [769].log_data[0].valid := 1, [769].log_data[1].valid := 1, [769].log_data[2].valid := 1, [769].log_data[3].valid := 1, [769].log_data[4].valid := 1, [769].log_data[5].valid := 1, [769].log_data[6].valid := 1, [769].log_data[7].valid := 1, [769].log_data[8].valid := 1, [769].log_data[9].valid := 1, [769].log_data[10].valid := 1, [769].log_data[11].valid := 1, [769].log_data[12].valid := 1, [769].log_data[13].valid := 1, [769].log_data[14].valid := 1, [769].log_data[15].valid := 1, [769].log_data[16].valid := 1, [769].log_data[17].valid := 1, [769].log_data[18].valid := 1, [769].log_data[19].valid := 1, [769].time.Year := 2023, [769].time.Month := 1, [769].time.Day := 12, [769].time.Hour := 8, [769].time.Minute := 29, [769].time.Second := 59, [770].log_data[0].min := 1.0, [770].log_data[0].max := 1.0, [770].log_data[0].total := 300.0, [770].log_data[0].time := 300.0, [770].log_data[0].minminute := 30, [770].log_data[0].maxminute := 30,
        [770].log_data[0].valid := 1, [770].log_data[1].valid := 1, [770].log_data[2].valid := 1, [770].log_data[3].valid := 1, [770].log_data[4].valid := 1, [770].log_data[5].valid := 1, [770].log_data[6].valid := 1, [770].log_data[7].valid := 1, [770].log_data[8].valid := 1, [770].log_data[9].valid := 1, [770].log_data[10].valid := 1, [770].log_data[11].valid := 1, [770].log_data[12].valid := 1, [770].log_data[13].valid := 1, [770].log_data[14].valid := 1, [770].log_data[15].valid := 1, [770].log_data[16].valid := 1, [770].log_data[17].valid := 1, [770].log_data[18].valid := 1, [770].log_data[19].valid := 1, [770].time.Year := 2023, [770].time.Month := 1, [770].time.Day := 12, [770].time.Hour := 8, [770].time.Minute := 34, [770].time.Second := 59, [771].log_data[0].min := 1.0, [771].log_data[0].max := 1.0, [771].log_data[0].total := 300.0, [771].log_data[0].time := 300.0, [771].log_data[0].minminute := 35, [771].log_data[0].maxminute := 35, [771].log_data[0].valid := 1, [771].log_data[1].valid := 1, [771].log_data[2].valid := 1, [771].log_data[3].valid := 1, [771].log_data[4].valid := 1, [771].log_data[5].valid := 1, [771].log_data[6].valid := 1, [771].log_data[7].valid := 1, [771].log_data[8].valid := 1, [771].log_data[9].valid := 1, [771].log_data[10].valid := 1, [771].log_data[11].valid := 1, [771].log_data[12].valid := 1, [771].log_data[13].valid := 1, [771].log_data[14].valid := 1, [771].log_data[15].valid := 1, [771].log_data[16].valid := 1, [771].log_data[17].valid := 1, [771].log_data[18].valid := 1, [771].log_data[19].valid := 1, [771].time.Year := 2023, [771].time.Month := 1, [771].time.Day := 12, [771].time.Hour := 8, [771].time.Minute := 39, [771].time.Second := 59, [772].log_data[0].min := 1.0, [772].log_data[0].max := 1.0,
        [772].log_data[0].total := 300.0, [772].log_data[0].time := 300.0, [772].log_data[0].minminute := 40, [772].log_data[0].maxminute := 40, [772].log_data[0].valid := 1, [772].log_data[1].valid := 1, [772].log_data[2].valid := 1, [772].log_data[3].valid := 1, [772].log_data[4].valid := 1, [772].log_data[5].valid := 1, [772].log_data[6].valid := 1, [772].log_data[7].valid := 1, [772].log_data[8].valid := 1, [772].log_data[9].valid := 1, [772].log_data[10].valid := 1, [772].log_data[11].valid := 1, [772].log_data[12].valid := 1, [772].log_data[13].valid := 1, [772].log_data[14].valid := 1, [772].log_data[15].valid := 1, [772].log_data[16].valid := 1, [772].log_data[17].valid := 1, [772].log_data[18].valid := 1, [772].log_data[19].valid := 1, [772].time.Year := 2023, [772].time.Month := 1, [772].time.Day := 12, [772].time.Hour := 8, [772].time.Minute := 44, [772].time.Second := 59, [773].log_data[0].min := 1.0, [773].log_data[0].max := 1.0, [773].log_data[0].total := 300.0, [773].log_data[0].time := 300.0, [773].log_data[0].minminute := 45, [773].log_data[0].maxminute := 45, [773].log_data[0].valid := 1, [773].log_data[1].valid := 1, [773].log_data[2].valid := 1, [773].log_data[3].valid := 1, [773].log_data[4].valid := 1, [773].log_data[5].valid := 1, [773].log_data[6].valid := 1, [773].log_data[7].valid := 1, [773].log_data[8].valid := 1, [773].log_data[9].valid := 1, [773].log_data[10].valid := 1, [773].log_data[11].valid := 1, [773].log_data[12].valid := 1, [773].log_data[13].valid := 1, [773].log_data[14].valid := 1, [773].log_data[15].valid := 1, [773].log_data[16].valid := 1, [773].log_data[17].valid := 1, [773].log_data[18].valid := 1, [773].log_data[19].valid := 1, [773].time.Year := 2023, [773].time.Month := 1, [773].time.Day := 12, [773].time.Hour := 8,
        [773].time.Minute := 49, [773].time.Second := 59, [774].log_data[0].min := 1.0, [774].log_data[0].max := 1.0, [774].log_data[0].total := 300.0, [774].log_data[0].time := 300.0, [774].log_data[0].minminute := 50, [774].log_data[0].maxminute := 50, [774].log_data[0].valid := 1, [774].log_data[1].valid := 1, [774].log_data[2].valid := 1, [774].log_data[3].valid := 1, [774].log_data[4].valid := 1, [774].log_data[5].valid := 1, [774].log_data[6].valid := 1, [774].log_data[7].valid := 1, [774].log_data[8].valid := 1, [774].log_data[9].valid := 1, [774].log_data[10].valid := 1, [774].log_data[11].valid := 1, [774].log_data[12].valid := 1, [774].log_data[13].valid := 1, [774].log_data[14].valid := 1, [774].log_data[15].valid := 1, [774].log_data[16].valid := 1, [774].log_data[17].valid := 1, [774].log_data[18].valid := 1, [774].log_data[19].valid := 1, [774].time.Year := 2023, [774].time.Month := 1, [774].time.Day := 12, [774].time.Hour := 8, [774].time.Minute := 54, [774].time.Second := 59, [775].log_data[0].min := 1.0, [775].log_data[0].max := 1.0, [775].log_data[0].total := 300.0, [775].log_data[0].time := 300.0, [775].log_data[0].minminute := 55, [775].log_data[0].maxminute := 55, [775].log_data[0].valid := 1, [775].log_data[1].valid := 1, [775].log_data[2].valid := 1, [775].log_data[3].valid := 1, [775].log_data[4].valid := 1, [775].log_data[5].valid := 1, [775].log_data[6].valid := 1, [775].log_data[7].valid := 1, [775].log_data[8].valid := 1, [775].log_data[9].valid := 1, [775].log_data[10].valid := 1, [775].log_data[11].valid := 1, [775].log_data[12].valid := 1, [775].log_data[13].valid := 1, [775].log_data[14].valid := 1, [775].log_data[15].valid := 1, [775].log_data[16].valid := 1, [775].log_data[17].valid := 1, [775].log_data[18].valid := 1, [775].log_data[19].valid := 1,
        [775].time.Year := 2023, [775].time.Month := 1, [775].time.Day := 12, [775].time.Hour := 8, [775].time.Minute := 59, [775].time.Second := 59, [776].log_data[0].min := 1.0, [776].log_data[0].max := 1.0, [776].log_data[0].total := 300.0, [776].log_data[0].time := 300.0, [776].log_data[0].valid := 1, [776].log_data[1].valid := 1, [776].log_data[2].valid := 1, [776].log_data[3].valid := 1, [776].log_data[4].valid := 1, [776].log_data[5].valid := 1, [776].log_data[6].valid := 1, [776].log_data[7].valid := 1, [776].log_data[8].valid := 1, [776].log_data[9].valid := 1, [776].log_data[10].valid := 1, [776].log_data[11].valid := 1, [776].log_data[12].valid := 1, [776].log_data[13].valid := 1, [776].log_data[14].valid := 1, [776].log_data[15].valid := 1, [776].log_data[16].valid := 1, [776].log_data[17].valid := 1, [776].log_data[18].valid := 1, [776].log_data[19].valid := 1, [776].time.Year := 2023, [776].time.Month := 1, [776].time.Day := 12, [776].time.Hour := 9, [776].time.Minute := 4, [776].time.Second := 59, [777].log_data[0].min := 1.0, [777].log_data[0].max := 1.0, [777].log_data[0].total := 300.0, [777].log_data[0].time := 300.0, [777].log_data[0].minminute := 5, [777].log_data[0].maxminute := 5, [777].log_data[0].valid := 1, [777].log_data[1].valid := 1, [777].log_data[2].valid := 1, [777].log_data[3].valid := 1, [777].log_data[4].valid := 1, [777].log_data[5].valid := 1, [777].log_data[6].valid := 1, [777].log_data[7].valid := 1, [777].log_data[8].valid := 1, [777].log_data[9].valid := 1, [777].log_data[10].valid := 1, [777].log_data[11].valid := 1, [777].log_data[12].valid := 1, [777].log_data[13].valid := 1, [777].log_data[14].valid := 1, [777].log_data[15].valid := 1, [777].log_data[16].valid := 1, [777].log_data[17].valid := 1,
        [777].log_data[18].valid := 1, [777].log_data[19].valid := 1, [777].time.Year := 2023, [777].time.Month := 1, [777].time.Day := 12, [777].time.Hour := 9, [777].time.Minute := 9, [777].time.Second := 59, [778].log_data[0].min := 1.0, [778].log_data[0].max := 1.0, [778].log_data[0].total := 300.0, [778].log_data[0].time := 300.0, [778].log_data[0].minminute := 10, [778].log_data[0].maxminute := 10, [778].log_data[0].valid := 1, [778].log_data[1].valid := 1, [778].log_data[2].valid := 1, [778].log_data[3].valid := 1, [778].log_data[4].valid := 1, [778].log_data[5].valid := 1, [778].log_data[6].valid := 1, [778].log_data[7].valid := 1, [778].log_data[8].valid := 1, [778].log_data[9].valid := 1, [778].log_data[10].valid := 1, [778].log_data[11].valid := 1, [778].log_data[12].valid := 1, [778].log_data[13].valid := 1, [778].log_data[14].valid := 1, [778].log_data[15].valid := 1, [778].log_data[16].valid := 1, [778].log_data[17].valid := 1, [778].log_data[18].valid := 1, [778].log_data[19].valid := 1, [778].time.Year := 2023, [778].time.Month := 1, [778].time.Day := 12, [778].time.Hour := 9, [778].time.Minute := 14, [778].time.Second := 59, [779].log_data[0].min := 1.0, [779].log_data[0].max := 1.0, [779].log_data[0].total := 300.0, [779].log_data[0].time := 300.0, [779].log_data[0].minminute := 15, [779].log_data[0].maxminute := 15, [779].log_data[0].valid := 1, [779].log_data[1].valid := 1, [779].log_data[2].valid := 1, [779].log_data[3].valid := 1, [779].log_data[4].valid := 1, [779].log_data[5].valid := 1, [779].log_data[6].valid := 1, [779].log_data[7].valid := 1, [779].log_data[8].valid := 1, [779].log_data[9].valid := 1, [779].log_data[10].valid := 1, [779].log_data[11].valid := 1, [779].log_data[12].valid := 1, [779].log_data[13].valid := 1,
        [779].log_data[14].valid := 1, [779].log_data[15].valid := 1, [779].log_data[16].valid := 1, [779].log_data[17].valid := 1, [779].log_data[18].valid := 1, [779].log_data[19].valid := 1, [779].time.Year := 2023, [779].time.Month := 1, [779].time.Day := 12, [779].time.Hour := 9, [779].time.Minute := 19, [779].time.Second := 59, [780].log_data[0].min := 1.0, [780].log_data[0].max := 1.0, [780].log_data[0].total := 300.0, [780].log_data[0].time := 300.0, [780].log_data[0].minminute := 20, [780].log_data[0].maxminute := 20, [780].log_data[0].valid := 1, [780].log_data[1].valid := 1, [780].log_data[2].valid := 1, [780].log_data[3].valid := 1, [780].log_data[4].valid := 1, [780].log_data[5].valid := 1, [780].log_data[6].valid := 1, [780].log_data[7].valid := 1, [780].log_data[8].valid := 1, [780].log_data[9].valid := 1, [780].log_data[10].valid := 1, [780].log_data[11].valid := 1, [780].log_data[12].valid := 1, [780].log_data[13].valid := 1, [780].log_data[14].valid := 1, [780].log_data[15].valid := 1, [780].log_data[16].valid := 1, [780].log_data[17].valid := 1, [780].log_data[18].valid := 1, [780].log_data[19].valid := 1, [780].time.Year := 2023, [780].time.Month := 1, [780].time.Day := 12, [780].time.Hour := 9, [780].time.Minute := 24, [780].time.Second := 59, [781].log_data[0].min := 1.0, [781].log_data[0].max := 1.0, [781].log_data[0].total := 300.0, [781].log_data[0].time := 300.0, [781].log_data[0].minminute := 25, [781].log_data[0].maxminute := 25, [781].log_data[0].valid := 1, [781].log_data[1].valid := 1, [781].log_data[2].valid := 1, [781].log_data[3].valid := 1, [781].log_data[4].valid := 1, [781].log_data[5].valid := 1, [781].log_data[6].valid := 1, [781].log_data[7].valid := 1, [781].log_data[8].valid := 1, [781].log_data[9].valid := 1,
        [781].log_data[10].valid := 1, [781].log_data[11].valid := 1, [781].log_data[12].valid := 1, [781].log_data[13].valid := 1, [781].log_data[14].valid := 1, [781].log_data[15].valid := 1, [781].log_data[16].valid := 1, [781].log_data[17].valid := 1, [781].log_data[18].valid := 1, [781].log_data[19].valid := 1, [781].time.Year := 2023, [781].time.Month := 1, [781].time.Day := 12, [781].time.Hour := 9, [781].time.Minute := 29, [781].time.Second := 59, [782].log_data[0].min := 1.0, [782].log_data[0].max := 1.0, [782].log_data[0].total := 300.0, [782].log_data[0].time := 300.0, [782].log_data[0].minminute := 30, [782].log_data[0].maxminute := 30, [782].log_data[0].valid := 1, [782].log_data[1].valid := 1, [782].log_data[2].valid := 1, [782].log_data[3].valid := 1, [782].log_data[4].valid := 1, [782].log_data[5].valid := 1, [782].log_data[6].valid := 1, [782].log_data[7].valid := 1, [782].log_data[8].valid := 1, [782].log_data[9].valid := 1, [782].log_data[10].valid := 1, [782].log_data[11].valid := 1, [782].log_data[12].valid := 1, [782].log_data[13].valid := 1, [782].log_data[14].valid := 1, [782].log_data[15].valid := 1, [782].log_data[16].valid := 1, [782].log_data[17].valid := 1, [782].log_data[18].valid := 1, [782].log_data[19].valid := 1, [782].time.Year := 2023, [782].time.Month := 1, [782].time.Day := 12, [782].time.Hour := 9, [782].time.Minute := 34, [782].time.Second := 59, [783].log_data[0].min := 1.0, [783].log_data[0].max := 1.0, [783].log_data[0].total := 300.0, [783].log_data[0].time := 300.0, [783].log_data[0].minminute := 35, [783].log_data[0].maxminute := 35, [783].log_data[0].valid := 1, [783].log_data[1].valid := 1, [783].log_data[2].valid := 1, [783].log_data[3].valid := 1, [783].log_data[4].valid := 1, [783].log_data[5].valid := 1,
